Yaskawa INFORM job: A_ROOF_UPPER_0614_2_PAINT_28.JBI

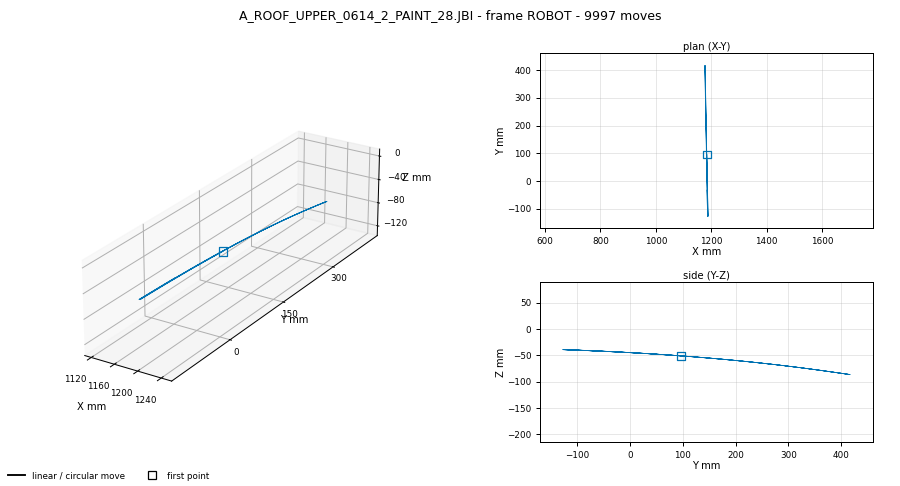
[picture p0: tool path of A_ROOF_UPPER_0614_2_PAINT_28.JBI in frame ROBOT, 9997 of 9997 moves have a stored position in this frame; points joined in program order, loops and branches not executed]
/JOB
//NAME A_ROOF_UPPER_0614_2_PAINT28
//POS
///NPOS 9997,0,0,0,0,0
///TOOL 1
///USER 0
///POSTYPE ROBOT
///RECTAN
///RCONF 1,0,0,0,0,0,0,0,0,0,0,0,0,0,0,0,0,0,0,0,0,0,0,0
C00000=1184.415,96.104,-50.756,-178.923,6.084,148.774
C00001=1184.420,95.856,-50.738,-178.925,6.082,148.774
C00002=1184.424,95.607,-50.720,-178.928,6.081,148.774
C00003=1184.429,95.357,-50.701,-178.931,6.080,148.775
C00004=1184.434,95.107,-50.683,-178.933,6.079,148.775
C00005=1184.439,94.858,-50.665,-178.936,6.078,148.776
C00006=1184.444,94.609,-50.647,-178.938,6.077,148.777
C00007=1184.449,94.360,-50.629,-178.941,6.076,148.777
C00008=1184.454,94.111,-50.611,-178.944,6.075,148.778
C00009=1184.458,93.861,-50.592,-178.947,6.073,148.778
C00010=1184.463,93.612,-50.574,-178.949,6.072,148.779
C00011=1184.468,93.362,-50.556,-178.952,6.071,148.779
C00012=1184.473,93.113,-50.538,-178.954,6.070,148.780
C00013=1184.478,92.864,-50.521,-178.957,6.068,148.780
C00014=1184.483,92.615,-50.503,-178.960,6.068,148.781
C00015=1184.488,92.366,-50.485,-178.962,6.066,148.781
C00016=1184.492,92.116,-50.466,-178.965,6.066,148.782
C00017=1184.497,91.867,-50.448,-178.968,6.064,148.782
C00018=1184.502,91.618,-50.430,-178.970,6.063,148.783
C00019=1184.507,91.368,-50.412,-178.973,6.062,148.783
C00020=1184.512,91.119,-50.394,-178.975,6.061,148.784
C00021=1184.517,90.869,-50.377,-178.978,6.060,148.784
C00022=1184.522,90.620,-50.359,-178.980,6.058,148.785
C00023=1184.527,90.371,-50.341,-178.983,6.058,148.785
C00024=1184.532,90.122,-50.323,-178.986,6.056,148.786
C00025=1184.537,89.873,-50.305,-178.988,6.056,148.787
C00026=1184.541,89.623,-50.287,-178.991,6.054,148.787
C00027=1184.546,89.374,-50.269,-178.994,6.053,148.788
C00028=1184.551,89.124,-50.252,-178.996,6.052,148.788
C00029=1184.556,88.875,-50.234,-178.999,6.051,148.789
C00030=1184.561,88.625,-50.216,-179.002,6.049,148.789
C00031=1184.566,88.376,-50.198,-179.004,6.049,148.790
C00032=1184.571,88.127,-50.180,-179.007,6.047,148.790
C00033=1184.576,87.877,-50.162,-179.010,6.046,148.791
C00034=1184.581,87.628,-50.144,-179.012,6.046,148.791
C00035=1184.586,87.379,-50.126,-179.015,6.044,148.792
C00036=1184.590,87.130,-50.109,-179.017,6.043,148.792
C00037=1184.595,86.881,-50.091,-179.020,6.042,148.793
C00038=1184.600,86.631,-50.074,-179.023,6.041,148.793
C00039=1184.605,86.382,-50.056,-179.025,6.039,148.794
C00040=1184.610,86.133,-50.038,-179.028,6.039,148.794
C00041=1184.615,85.883,-50.021,-179.031,6.037,148.795
C00042=1184.620,85.634,-50.003,-179.033,6.036,148.796
C00043=1184.625,85.385,-49.985,-179.035,6.036,148.796
C00044=1184.629,85.136,-49.967,-179.039,6.034,148.797
C00045=1184.634,84.886,-49.950,-179.041,6.033,148.797
C00046=1184.639,84.637,-49.932,-179.044,6.032,148.798
C00047=1184.644,84.388,-49.914,-179.046,6.031,148.798
C00048=1184.649,84.138,-49.897,-179.049,6.030,148.799
C00049=1184.654,83.889,-49.879,-179.051,6.029,148.799
C00050=1184.659,83.639,-49.862,-179.054,6.028,148.800
C00051=1184.664,83.390,-49.844,-179.057,6.027,148.800
C00052=1184.669,83.141,-49.826,-179.059,6.026,148.801
C00053=1184.674,82.891,-49.809,-179.062,6.024,148.801
C00054=1184.678,82.642,-49.791,-179.065,6.024,148.802
C00055=1184.683,82.392,-49.774,-179.067,6.023,148.802
C00056=1184.688,82.143,-49.756,-179.070,6.021,148.803
C00057=1184.693,81.894,-49.738,-179.072,6.021,148.803
C00058=1184.698,81.645,-49.722,-179.075,6.019,148.804
C00059=1184.702,81.395,-49.704,-179.078,6.018,148.805
C00060=1184.708,81.146,-49.686,-179.081,6.017,148.805
C00061=1184.713,80.877,-49.667,-179.083,6.016,148.806
C00062=1184.719,80.609,-49.649,-179.086,6.015,148.806
C00063=1184.723,80.341,-49.630,-179.089,6.014,148.807
C00064=1184.728,80.072,-49.611,-179.092,6.013,148.808
C00065=1184.734,79.823,-49.594,-179.094,6.012,148.808
C00066=1184.739,79.573,-49.576,-179.097,6.011,148.809
C00067=1184.743,79.324,-49.559,-179.099,6.010,148.809
C00068=1184.749,79.075,-49.542,-179.102,6.009,148.810
C00069=1184.754,78.826,-49.524,-179.105,6.007,148.810
C00070=1184.758,78.576,-49.508,-179.107,6.007,148.811
C00071=1184.763,78.327,-49.490,-179.110,6.005,148.811
C00072=1184.768,78.077,-49.472,-179.113,6.005,148.812
C00073=1184.773,77.828,-49.455,-179.115,6.004,148.812
C00074=1184.778,77.579,-49.438,-179.118,6.002,148.813
C00075=1184.783,77.329,-49.420,-179.120,6.001,148.813
C00076=1184.788,77.081,-49.403,-179.123,6.000,148.814
C00077=1184.793,76.831,-49.386,-179.126,5.999,148.814
C00078=1184.797,76.582,-49.369,-179.128,5.999,148.815
C00079=1184.802,76.332,-49.351,-179.131,5.997,148.816
C00080=1184.808,76.082,-49.334,-179.134,5.996,148.816
C00081=1184.812,75.833,-49.317,-179.136,5.995,148.817
C00082=1184.817,75.584,-49.300,-179.139,5.994,148.817
C00083=1184.822,75.335,-49.283,-179.141,5.993,148.818
C00084=1184.827,75.085,-49.266,-179.144,5.992,148.818
C00085=1184.831,74.836,-49.249,-179.146,5.991,148.819
C00086=1184.837,74.586,-49.231,-179.149,5.990,148.819
C00087=1184.842,74.337,-49.214,-179.152,5.989,148.820
C00088=1184.846,74.088,-49.197,-179.154,5.988,148.821
C00089=1184.852,73.839,-49.180,-179.157,5.988,148.821
C00090=1184.856,73.589,-49.163,-179.160,5.986,148.822
C00091=1184.862,73.339,-49.146,-179.162,5.985,148.822
C00092=1184.866,73.091,-49.128,-179.165,5.984,148.823
C00093=1184.871,72.841,-49.111,-179.168,5.983,148.823
C00094=1184.876,72.592,-49.095,-179.170,5.982,148.824
C00095=1184.881,72.342,-49.078,-179.173,5.981,148.824
C00096=1184.886,72.093,-49.061,-179.175,5.980,148.825
C00097=1184.891,71.843,-49.044,-179.178,5.979,148.826
C00098=1184.896,71.595,-49.027,-179.181,5.978,148.826
C00099=1184.901,71.345,-49.009,-179.183,5.977,148.827
C00100=1184.905,71.095,-48.993,-179.186,5.977,148.827
C00101=1184.911,70.846,-48.976,-179.189,5.975,148.828
C00102=1184.915,70.596,-48.959,-179.191,5.974,148.828
C00103=1184.921,70.347,-48.942,-179.193,5.974,148.829
C00104=1184.925,70.098,-48.925,-179.197,5.972,148.829
C00105=1184.930,69.848,-48.907,-179.199,5.971,148.830
C00106=1184.935,69.599,-48.891,-179.201,5.971,148.831
C00107=1184.940,69.350,-48.874,-179.204,5.969,148.831
C00108=1184.945,69.100,-48.857,-179.207,5.969,148.832
C00109=1184.950,68.851,-48.840,-179.209,5.968,148.832
C00110=1184.955,68.602,-48.823,-179.212,5.966,148.833
C00111=1184.960,68.352,-48.807,-179.215,5.966,148.833
C00112=1184.964,68.103,-48.790,-179.217,5.965,148.834
C00113=1184.970,67.853,-48.773,-179.220,5.964,148.835
C00114=1184.975,67.604,-48.757,-179.222,5.963,148.835
C00115=1184.980,67.354,-48.739,-179.225,5.962,148.836
C00116=1184.984,67.105,-48.723,-179.228,5.960,148.836
C00117=1184.990,66.856,-48.706,-179.230,5.960,148.837
C00118=1184.995,66.606,-48.689,-179.233,5.959,148.837
C00119=1184.999,66.357,-48.672,-179.236,5.958,148.838
C00120=1185.004,66.107,-48.656,-179.238,5.957,148.838
C00121=1185.010,65.858,-48.639,-179.240,5.956,148.839
C00122=1185.014,65.609,-48.622,-179.244,5.955,148.840
C00123=1185.018,65.359,-48.605,-179.246,5.954,148.840
C00124=1185.024,65.110,-48.589,-179.248,5.953,148.841
C00125=1185.029,64.861,-48.572,-179.252,5.952,148.841
C00126=1185.033,64.611,-48.555,-179.254,5.951,148.842
C00127=1185.039,64.362,-48.538,-179.256,5.951,148.842
C00128=1185.044,64.112,-48.522,-179.258,5.950,148.843
C00129=1185.049,63.863,-48.506,-179.262,5.948,148.843
C00130=1185.053,63.614,-48.489,-179.264,5.948,148.844
C00131=1185.059,63.364,-48.472,-179.266,5.947,148.845
C00132=1185.064,63.115,-48.456,-179.270,5.946,148.845
C00133=1185.068,62.866,-48.439,-179.272,5.945,148.846
C00134=1185.073,62.616,-48.423,-179.274,5.944,148.846
C00135=1185.079,62.367,-48.406,-179.277,5.943,148.847
C00136=1185.083,62.117,-48.390,-179.280,5.942,148.847
C00137=1185.088,61.868,-48.373,-179.282,5.941,148.848
C00138=1185.093,61.619,-48.357,-179.285,5.941,148.849
C00139=1185.098,61.369,-48.339,-179.288,5.939,148.849
C00140=1185.103,61.120,-48.324,-179.290,5.938,148.850
C00141=1185.108,60.870,-48.307,-179.293,5.938,148.850
C00142=1185.113,60.621,-48.291,-179.295,5.936,148.851
C00143=1185.117,60.372,-48.274,-179.298,5.936,148.851
C00144=1185.123,60.121,-48.258,-179.301,5.935,148.852
C00145=1185.128,59.873,-48.241,-179.303,5.934,148.853
C00146=1185.133,59.623,-48.225,-179.306,5.933,148.853
C00147=1185.138,59.374,-48.208,-179.308,5.932,148.854
C00148=1185.142,59.124,-48.192,-179.311,5.931,148.854
C00149=1185.148,58.875,-48.176,-179.313,5.931,148.855
C00150=1185.153,58.626,-48.159,-179.316,5.929,148.855
C00151=1185.158,58.376,-48.143,-179.319,5.929,148.856
C00152=1185.163,58.127,-48.127,-179.321,5.928,148.856
C00153=1185.167,57.877,-48.110,-179.324,5.927,148.857
C00154=1185.172,57.628,-48.094,-179.327,5.926,148.858
C00155=1185.177,57.378,-48.078,-179.329,5.925,148.858
C00156=1185.182,57.130,-48.061,-179.332,5.925,148.859
C00157=1185.188,56.879,-48.045,-179.334,5.923,148.859
C00158=1185.193,56.630,-48.029,-179.337,5.922,148.860
C00159=1185.197,56.380,-48.013,-179.340,5.922,148.861
C00160=1185.202,56.132,-47.996,-179.342,5.921,148.861
C00161=1185.207,55.882,-47.980,-179.345,5.920,148.862
C00162=1185.212,55.633,-47.964,-179.347,5.919,148.862
C00163=1185.217,55.383,-47.947,-179.350,5.918,148.863
C00164=1185.222,55.134,-47.932,-179.352,5.918,148.864
C00165=1185.227,54.865,-47.914,-179.355,5.916,148.864
C00166=1185.232,54.597,-47.897,-179.358,5.915,148.865
C00167=1185.238,54.328,-47.880,-179.361,5.914,148.865
C00168=1185.243,54.059,-47.861,-179.364,5.914,148.866
C00169=1185.249,53.810,-47.845,-179.366,5.913,148.866
C00170=1185.253,53.560,-47.829,-179.369,5.911,148.867
C00171=1185.259,53.311,-47.813,-179.372,5.911,148.868
C00172=1185.264,53.062,-47.797,-179.374,5.910,148.868
C00173=1185.269,52.812,-47.781,-179.376,5.909,148.869
C00174=1185.274,52.563,-47.765,-179.379,5.908,148.869
C00175=1185.278,52.313,-47.749,-179.382,5.907,148.870
C00176=1185.284,52.064,-47.733,-179.384,5.907,148.871
C00177=1185.288,51.814,-47.716,-179.386,5.906,148.871
C00178=1185.294,51.565,-47.701,-179.389,5.905,148.872
C00179=1185.298,51.316,-47.684,-179.392,5.904,148.872
C00180=1185.303,51.066,-47.668,-179.395,5.903,148.873
C00181=1185.308,50.818,-47.653,-179.397,5.903,148.874
C00182=1185.313,50.568,-47.637,-179.399,5.902,148.874
C00183=1185.318,50.318,-47.621,-179.403,5.900,148.875
C00184=1185.322,50.069,-47.605,-179.405,5.900,148.875
C00185=1185.328,49.819,-47.589,-179.407,5.899,148.876
C00186=1185.332,49.570,-47.572,-179.410,5.898,148.876
C00187=1185.338,49.320,-47.557,-179.413,5.898,148.877
C00188=1185.343,49.071,-47.541,-179.415,5.896,148.878
C00189=1185.348,48.822,-47.524,-179.418,5.896,148.878
C00190=1185.353,48.572,-47.509,-179.420,5.895,148.879
C00191=1185.358,48.322,-47.493,-179.423,5.894,148.879
C00192=1185.362,48.073,-47.478,-179.426,5.893,148.880
C00193=1185.368,47.824,-47.462,-179.428,5.892,148.880
C00194=1185.372,47.574,-47.446,-179.431,5.892,148.881
C00195=1185.378,47.325,-47.430,-179.433,5.891,148.882
C00196=1185.383,47.076,-47.414,-179.436,5.890,148.882
C00197=1185.388,46.826,-47.398,-179.439,5.889,148.883
C00198=1185.393,46.576,-47.382,-179.441,5.888,148.883
C00199=1185.398,46.326,-47.366,-179.444,5.888,148.884
C00200=1185.402,46.078,-47.351,-179.446,5.887,148.885
C00201=1185.407,45.828,-47.335,-179.448,5.886,148.885
C00202=1185.412,45.578,-47.319,-179.452,5.885,148.886
C00203=1185.418,45.329,-47.303,-179.454,5.884,148.886
C00204=1185.423,45.079,-47.288,-179.456,5.883,148.887
C00205=1185.427,44.830,-47.272,-179.459,5.883,148.888
C00206=1185.432,44.581,-47.256,-179.462,5.882,148.888
C00207=1185.438,44.331,-47.241,-179.464,5.881,148.889
C00208=1185.442,44.081,-47.225,-179.467,5.880,148.889
C00209=1185.448,43.832,-47.209,-179.469,5.879,148.890
C00210=1185.452,43.583,-47.194,-179.472,5.879,148.890
C00211=1185.457,43.334,-47.178,-179.474,5.878,148.891
C00212=1185.462,43.084,-47.162,-179.477,5.877,148.892
C00213=1185.468,42.835,-47.146,-179.480,5.876,148.892
C00214=1185.472,42.585,-47.131,-179.482,5.876,148.893
C00215=1185.477,42.335,-47.115,-179.485,5.875,148.893
C00216=1185.482,42.086,-47.100,-179.487,5.874,148.894
C00217=1185.488,41.837,-47.084,-179.490,5.874,148.895
C00218=1185.492,41.587,-47.069,-179.493,5.872,148.895
C00219=1185.497,41.337,-47.053,-179.495,5.871,148.896
C00220=1185.503,41.088,-47.038,-179.498,5.871,148.896
C00221=1185.508,40.839,-47.021,-179.500,5.870,148.897
C00222=1185.512,40.589,-47.006,-179.503,5.870,148.898
C00223=1185.517,40.340,-46.990,-179.505,5.869,148.898
C00224=1185.523,40.091,-46.975,-179.508,5.867,148.899
C00225=1185.527,39.842,-46.960,-179.511,5.867,148.899
C00226=1185.532,39.591,-46.944,-179.513,5.866,148.900
C00227=1185.537,39.342,-46.928,-179.516,5.865,148.900
C00228=1185.542,39.093,-46.913,-179.518,5.865,148.901
C00229=1185.547,38.844,-46.898,-179.520,5.864,148.902
C00230=1185.553,38.594,-46.882,-179.523,5.864,148.902
C00231=1185.557,38.344,-46.867,-179.526,5.862,148.903
C00232=1185.563,38.094,-46.852,-179.528,5.861,148.903
C00233=1185.568,37.845,-46.836,-179.531,5.861,148.904
C00234=1185.573,37.596,-46.821,-179.534,5.860,148.905
C00235=1185.577,37.346,-46.805,-179.536,5.860,148.905
C00236=1185.582,37.097,-46.790,-179.538,5.859,148.906
C00237=1185.587,36.847,-46.775,-179.542,5.858,148.907
C00238=1185.593,36.598,-46.759,-179.544,5.857,148.907
C00239=1185.597,36.349,-46.744,-179.546,5.856,148.908
C00240=1185.603,36.099,-46.729,-179.549,5.856,148.908
C00241=1185.607,35.850,-46.713,-179.551,5.855,148.909
C00242=1185.613,35.599,-46.698,-179.554,5.854,148.909
C00243=1185.618,35.350,-46.683,-179.557,5.854,148.910
C00244=1185.623,35.101,-46.668,-179.559,5.852,148.911
C00245=1185.628,34.852,-46.652,-179.562,5.852,148.911
C00246=1185.632,34.602,-46.637,-179.565,5.851,148.912
C00247=1185.637,34.352,-46.621,-179.567,5.850,148.912
C00248=1185.642,34.103,-46.607,-179.569,5.850,148.913
C00249=1185.648,33.853,-46.591,-179.572,5.849,148.914
C00250=1185.652,33.604,-46.576,-179.574,5.848,148.914
C00251=1185.658,33.355,-46.561,-179.577,5.848,148.915
C00252=1185.662,33.106,-46.546,-179.580,5.847,148.916
C00253=1185.668,32.855,-46.530,-179.582,5.846,148.916
C00254=1185.672,32.606,-46.515,-179.585,5.845,148.917
C00255=1185.678,32.356,-46.500,-179.588,5.845,148.917
C00256=1185.682,32.107,-46.485,-179.590,5.844,148.918
C00257=1185.688,31.857,-46.470,-179.592,5.843,148.918
C00258=1185.693,31.608,-46.455,-179.595,5.843,148.919
C00259=1185.698,31.359,-46.439,-179.597,5.842,148.920
C00260=1185.703,31.110,-46.424,-179.600,5.841,148.920
C00261=1185.708,30.860,-46.410,-179.603,5.840,148.921
C00262=1185.712,30.610,-46.394,-179.605,5.839,148.921
C00263=1185.718,30.361,-46.379,-179.608,5.839,148.922
C00264=1185.723,30.111,-46.364,-179.610,5.838,148.923
C00265=1185.728,29.861,-46.349,-179.613,5.838,148.923
C00266=1185.733,29.612,-46.334,-179.615,5.837,148.924
C00267=1185.738,29.363,-46.320,-179.618,5.836,148.925
C00268=1185.743,29.113,-46.304,-179.621,5.836,148.925
C00269=1185.748,28.844,-46.288,-179.623,5.834,148.926
C00270=1185.754,28.575,-46.272,-179.626,5.834,148.926
C00271=1185.759,28.307,-46.255,-179.629,5.833,148.927
C00272=1185.765,28.038,-46.239,-179.631,5.833,148.928
C00273=1185.770,27.788,-46.225,-179.634,5.831,148.928
C00274=1185.775,27.539,-46.209,-179.637,5.831,148.929
C00275=1185.780,27.290,-46.194,-179.639,5.830,148.930
C00276=1185.785,27.040,-46.180,-179.642,5.830,148.930
C00277=1185.790,26.791,-46.164,-179.645,5.829,148.931
C00278=1185.795,26.541,-46.150,-179.647,5.828,148.931
C00279=1185.800,26.292,-46.135,-179.649,5.828,148.932
C00280=1185.805,26.042,-46.120,-179.652,5.827,148.933
C00281=1185.810,25.793,-46.105,-179.654,5.826,148.933
C00282=1185.815,25.543,-46.091,-179.657,5.826,148.934
C00283=1185.820,25.294,-46.075,-179.659,5.825,148.934
C00284=1185.825,25.044,-46.061,-179.662,5.824,148.935
C00285=1185.830,24.795,-46.046,-179.665,5.823,148.936
C00286=1185.836,24.545,-46.031,-179.667,5.823,148.936
C00287=1185.840,24.296,-46.016,-179.670,5.822,148.937
C00288=1185.845,24.046,-46.002,-179.672,5.821,148.937
C00289=1185.851,23.797,-45.986,-179.675,5.821,148.938
C00290=1185.856,23.547,-45.972,-179.678,5.820,148.939
C00291=1185.860,23.298,-45.957,-179.680,5.820,148.939
C00292=1185.865,23.048,-45.943,-179.682,5.819,148.940
C00293=1185.871,22.798,-45.928,-179.685,5.819,148.941
C00294=1185.876,22.549,-45.913,-179.687,5.818,148.941
C00295=1185.880,22.299,-45.899,-179.690,5.817,148.942
C00296=1185.885,22.050,-45.884,-179.692,5.817,148.942
C00297=1185.891,21.800,-45.869,-179.695,5.816,148.943
C00298=1185.896,21.551,-45.855,-179.698,5.815,148.944
C00299=1185.900,21.301,-45.840,-179.701,5.814,148.944
C00300=1185.905,21.052,-45.825,-179.703,5.814,148.945
C00301=1185.911,20.802,-45.810,-179.705,5.813,148.945
C00302=1185.916,20.553,-45.796,-179.708,5.812,148.946
C00303=1185.921,20.303,-45.781,-179.711,5.812,148.947
C00304=1185.925,20.054,-45.766,-179.713,5.811,148.947
C00305=1185.930,19.804,-45.752,-179.715,5.810,148.948
C00306=1185.936,19.554,-45.737,-179.718,5.810,148.949
C00307=1185.941,19.304,-45.723,-179.720,5.809,148.949
C00308=1185.946,19.055,-45.708,-179.723,5.808,148.950
C00309=1185.951,18.806,-45.694,-179.726,5.808,148.950
C00310=1185.956,18.557,-45.680,-179.728,5.807,148.951
C00311=1185.961,18.308,-45.665,-179.730,5.807,148.951
C00312=1185.966,18.057,-45.650,-179.733,5.806,148.952
C00313=1185.971,17.808,-45.635,-179.736,5.806,148.953
C00314=1185.976,17.558,-45.621,-179.738,5.805,148.953
C00315=1185.981,17.309,-45.606,-179.740,5.804,148.954
C00316=1185.986,17.059,-45.592,-179.743,5.804,148.955
C00317=1185.991,16.810,-45.578,-179.745,5.803,148.955
C00318=1185.996,16.560,-45.563,-179.749,5.802,148.956
C00319=1186.002,16.311,-45.549,-179.751,5.801,148.956
C00320=1186.007,16.061,-45.534,-179.754,5.801,148.957
C00321=1186.012,15.812,-45.520,-179.756,5.800,148.958
C00322=1186.017,15.562,-45.505,-179.759,5.799,148.958
C00323=1186.022,15.312,-45.491,-179.761,5.799,148.959
C00324=1186.027,15.063,-45.477,-179.763,5.798,148.959
C00325=1186.031,14.813,-45.462,-179.766,5.797,148.960
C00326=1186.037,14.564,-45.448,-179.769,5.797,148.961
C00327=1186.042,14.315,-45.434,-179.771,5.796,148.962
C00328=1186.047,14.065,-45.419,-179.774,5.796,148.962
C00329=1186.052,13.815,-45.405,-179.776,5.795,148.963
C00330=1186.057,13.566,-45.391,-179.779,5.795,148.963
C00331=1186.062,13.316,-45.376,-179.781,5.794,148.964
C00332=1186.067,13.067,-45.363,-179.784,5.793,148.964
C00333=1186.073,12.817,-45.348,-179.786,5.793,148.965
C00334=1186.077,12.568,-45.333,-179.789,5.792,148.966
C00335=1186.082,12.318,-45.318,-179.791,5.791,148.966
C00336=1186.087,12.068,-45.304,-179.794,5.791,148.967
C00337=1186.093,11.819,-45.290,-179.796,5.791,148.968
C00338=1186.098,11.570,-45.276,-179.799,5.790,148.968
C00339=1186.103,11.320,-45.262,-179.801,5.789,148.969
C00340=1186.108,11.070,-45.247,-179.804,5.789,148.969
C00341=1186.113,10.821,-45.233,-179.807,5.788,148.970
C00342=1186.118,10.572,-45.219,-179.809,5.787,148.971
C00343=1186.123,10.322,-45.206,-179.811,5.787,148.971
C00344=1186.128,10.072,-45.191,-179.814,5.786,148.972
C00345=1186.132,9.823,-45.177,-179.816,5.786,148.972
C00346=1186.138,9.574,-45.163,-179.819,5.785,148.973
C00347=1186.143,9.324,-45.149,-179.821,5.785,148.974
C00348=1186.148,9.074,-45.135,-179.824,5.784,148.975
C00349=1186.153,8.825,-45.120,-179.826,5.783,148.975
C00350=1186.158,8.575,-45.106,-179.829,5.783,148.976
C00351=1186.163,8.326,-45.092,-179.832,5.782,148.976
C00352=1186.169,8.076,-45.078,-179.834,5.781,148.977
C00353=1186.174,7.826,-45.064,-179.836,5.781,148.977
C00354=1186.179,7.577,-45.050,-179.839,5.780,148.978
C00355=1186.184,7.327,-45.036,-179.842,5.780,148.979
C00356=1186.189,7.077,-45.022,-179.844,5.779,148.979
C00357=1186.193,6.828,-45.008,-179.847,5.779,148.980
C00358=1186.199,6.579,-44.994,-179.849,5.778,148.981
C00359=1186.204,6.329,-44.980,-179.852,5.778,148.981
C00360=1186.209,6.080,-44.966,-179.854,5.777,148.982
C00361=1186.214,5.829,-44.952,-179.857,5.776,148.983
C00362=1186.220,5.580,-44.938,-179.859,5.776,148.983
C00363=1186.225,5.330,-44.924,-179.861,5.775,148.984
C00364=1186.229,5.081,-44.910,-179.864,5.774,148.984
C00365=1186.234,4.832,-44.896,-179.867,5.774,148.985
C00366=1186.239,4.582,-44.882,-179.869,5.774,148.986
C00367=1186.245,4.332,-44.868,-179.872,5.773,148.986
C00368=1186.250,4.083,-44.855,-179.874,5.772,148.987
C00369=1186.255,3.833,-44.840,-179.877,5.772,148.988
C00370=1186.259,3.584,-44.827,-179.880,5.771,148.988
C00371=1186.265,3.335,-44.813,-179.882,5.770,148.989
C00372=1186.270,3.085,-44.799,-179.884,5.770,148.989
C00373=1186.275,2.815,-44.784,-179.887,5.769,148.990
C00374=1186.281,2.546,-44.769,-179.890,5.769,148.991
C00375=1186.287,2.278,-44.754,-179.892,5.768,148.991
C00376=1186.292,2.008,-44.739,-179.895,5.768,148.992
C00377=1186.297,1.758,-44.725,-179.897,5.767,148.993
C00378=1186.302,1.509,-44.712,-179.900,5.767,148.993
C00379=1186.307,1.260,-44.698,-179.902,5.766,148.994
C00380=1186.312,1.009,-44.684,-179.905,5.766,148.995
C00381=1186.318,0.760,-44.670,-179.907,5.765,148.995
C00382=1186.322,0.511,-44.656,-179.910,5.764,148.996
C00383=1186.327,0.260,-44.643,-179.913,5.764,148.997
C00384=1186.333,0.011,-44.629,-179.915,5.763,148.997
C00385=1186.338,-0.238,-44.615,-179.917,5.763,148.998
C00386=1186.342,-0.488,-44.602,-179.920,5.762,148.998
C00387=1186.348,-0.737,-44.588,-179.922,5.762,148.999
C00388=1186.353,-0.987,-44.574,-179.925,5.762,149.000
C00389=1186.358,-1.236,-44.561,-179.927,5.761,149.000
C00390=1186.363,-1.486,-44.547,-179.930,5.761,149.001
C00391=1186.368,-1.736,-44.532,-179.932,5.760,149.002
C00392=1186.373,-1.985,-44.520,-179.934,5.759,149.002
C00393=1186.378,-2.235,-44.506,-179.937,5.759,149.003
C00394=1186.384,-2.484,-44.492,-179.940,5.758,149.003
C00395=1186.388,-2.734,-44.479,-179.942,5.758,149.004
C00396=1186.394,-2.983,-44.465,-179.945,5.757,149.005
C00397=1186.399,-3.233,-44.451,-179.947,5.757,149.005
C00398=1186.403,-3.483,-44.437,-179.950,5.756,149.006
C00399=1186.409,-3.732,-44.424,-179.953,5.756,149.007
C00400=1186.414,-3.982,-44.410,-179.955,5.755,149.007
C00401=1186.419,-4.231,-44.397,-179.957,5.754,149.008
C00402=1186.424,-4.481,-44.383,-179.960,5.754,149.008
C00403=1186.430,-4.731,-44.370,-179.962,5.754,149.009
C00404=1186.434,-4.980,-44.356,-179.964,5.753,149.010
C00405=1186.440,-5.230,-44.343,-179.967,5.753,149.010
C00406=1186.444,-5.479,-44.329,-179.970,5.752,149.011
C00407=1186.449,-5.729,-44.316,-179.972,5.752,149.011
C00408=1186.455,-5.978,-44.302,-179.974,5.751,149.012
C00409=1186.460,-6.228,-44.289,-179.977,5.751,149.013
C00410=1186.465,-6.478,-44.276,-179.980,5.750,149.014
C00411=1186.470,-6.727,-44.262,-179.982,5.749,149.014
C00412=1186.476,-6.977,-44.249,-179.985,5.749,149.015
C00413=1186.480,-7.227,-44.235,-179.987,5.748,149.015
C00414=1186.486,-7.476,-44.222,-179.990,5.748,149.016
C00415=1186.491,-7.726,-44.208,-179.992,5.747,149.017
C00416=1186.496,-7.975,-44.195,-179.994,5.747,149.017
C00417=1186.501,-8.225,-44.182,-179.997,5.747,149.018
C00418=1186.506,-8.474,-44.168,-179.999,5.746,149.019
C00419=1186.511,-8.724,-44.155,179.998,5.746,149.019
C00420=1186.516,-8.973,-44.141,179.996,5.745,149.020
C00421=1186.521,-9.223,-44.128,179.993,5.745,149.020
C00422=1186.526,-9.473,-44.115,179.990,5.744,149.021
C00423=1186.531,-9.722,-44.101,179.988,5.743,149.022
C00424=1186.536,-9.972,-44.088,179.986,5.743,149.022
C00425=1186.542,-10.222,-44.075,179.983,5.742,149.023
C00426=1186.546,-10.471,-44.061,179.981,5.743,149.024
C00427=1186.552,-10.720,-44.048,179.979,5.742,149.024
C00428=1186.557,-10.970,-44.035,179.976,5.741,149.025
C00429=1186.562,-11.219,-44.021,179.973,5.741,149.026
C00430=1186.567,-11.469,-44.008,179.971,5.740,149.026
C00431=1186.573,-11.719,-43.995,179.969,5.740,149.027
C00432=1186.577,-11.969,-43.982,179.966,5.739,149.027
C00433=1186.583,-12.218,-43.968,179.963,5.739,149.028
C00434=1186.587,-12.468,-43.955,179.961,5.738,149.029
C00435=1186.592,-12.717,-43.943,179.958,5.737,149.029
C00436=1186.598,-12.967,-43.930,179.956,5.738,149.030
C00437=1186.602,-13.216,-43.916,179.954,5.737,149.031
C00438=1186.608,-13.466,-43.903,179.952,5.736,149.031
C00439=1186.613,-13.716,-43.890,179.949,5.736,149.032
C00440=1186.619,-13.966,-43.877,179.946,5.735,149.032
C00441=1186.624,-14.214,-43.863,179.944,5.735,149.033
C00442=1186.628,-14.464,-43.850,179.941,5.734,149.034
C00443=1186.634,-14.714,-43.837,179.939,5.734,149.034
C00444=1186.638,-14.964,-43.824,179.937,5.734,149.035
C00445=1186.644,-15.213,-43.811,179.934,5.734,149.036
C00446=1186.649,-15.463,-43.798,179.932,5.733,149.036
C00447=1186.654,-15.712,-43.785,179.929,5.732,149.037
C00448=1186.660,-15.962,-43.771,179.927,5.732,149.038
C00449=1186.664,-16.212,-43.758,179.924,5.731,149.038
C00450=1186.669,-16.461,-43.746,179.922,5.731,149.039
C00451=1186.675,-16.711,-43.733,179.919,5.730,149.039
C00452=1186.680,-16.961,-43.720,179.917,5.730,149.040
C00453=1186.685,-17.210,-43.707,179.914,5.730,149.041
C00454=1186.691,-17.460,-43.694,179.912,5.729,149.041
C00455=1186.695,-17.709,-43.680,179.909,5.729,149.042
C00456=1186.700,-17.959,-43.668,179.907,5.728,149.043
C00457=1186.706,-18.208,-43.654,179.904,5.728,149.043
C00458=1186.710,-18.458,-43.641,179.902,5.727,149.044
C00459=1186.715,-18.708,-43.629,179.899,5.726,149.045
C00460=1186.721,-18.957,-43.616,179.897,5.727,149.045
C00461=1186.726,-19.207,-43.603,179.895,5.726,149.046
C00462=1186.731,-19.457,-43.590,179.892,5.725,149.046
C00463=1186.736,-19.706,-43.577,179.890,5.725,149.047
C00464=1186.741,-19.956,-43.564,179.887,5.725,149.048
C00465=1186.746,-20.206,-43.551,179.885,5.724,149.048
C00466=1186.752,-20.455,-43.539,179.882,5.723,149.049
C00467=1186.757,-20.705,-43.525,179.880,5.724,149.050
C00468=1186.762,-20.955,-43.513,179.878,5.723,149.050
C00469=1186.767,-21.204,-43.500,179.875,5.722,149.051
C00470=1186.772,-21.454,-43.487,179.873,5.722,149.051
C00471=1186.777,-21.704,-43.474,179.870,5.721,149.052
C00472=1186.783,-21.953,-43.461,179.867,5.721,149.053
C00473=1186.788,-22.202,-43.449,179.866,5.721,149.053
C00474=1186.792,-22.452,-43.436,179.863,5.720,149.054
C00475=1186.798,-22.702,-43.422,179.860,5.720,149.055
C00476=1186.803,-22.951,-43.410,179.858,5.720,149.055
C00477=1186.808,-23.221,-43.396,179.855,5.719,149.056
C00478=1186.814,-23.491,-43.382,179.852,5.719,149.057
C00479=1186.820,-23.761,-43.369,179.850,5.718,149.058
C00480=1186.825,-24.030,-43.356,179.847,5.718,149.058
C00481=1186.831,-24.280,-43.342,179.845,5.717,149.059
C00482=1186.836,-24.529,-43.330,179.842,5.716,149.059
C00483=1186.840,-24.779,-43.317,179.840,5.717,149.060
C00484=1186.845,-25.029,-43.304,179.838,5.716,149.061
C00485=1186.851,-25.278,-43.292,179.835,5.715,149.061
C00486=1186.856,-25.527,-43.279,179.833,5.715,149.062
C00487=1186.861,-25.778,-43.266,179.830,5.715,149.063
C00488=1186.866,-26.028,-43.254,179.828,5.714,149.063
C00489=1186.872,-26.277,-43.241,179.826,5.714,149.064
C00490=1186.877,-26.526,-43.228,179.823,5.714,149.064
C00491=1186.881,-26.776,-43.215,179.821,5.713,149.065
C00492=1186.886,-27.025,-43.203,179.818,5.712,149.066
C00493=1186.892,-27.275,-43.191,179.816,5.712,149.066
C00494=1186.897,-27.525,-43.178,179.813,5.711,149.067
C00495=1186.903,-27.774,-43.165,179.811,5.712,149.068
C00496=1186.907,-28.024,-43.152,179.809,5.711,149.068
C00497=1186.913,-28.274,-43.140,179.806,5.710,149.069
C00498=1186.918,-28.524,-43.128,179.803,5.710,149.070
C00499=1186.923,-28.773,-43.115,179.801,5.710,149.070
C00500=1186.928,-29.022,-43.102,179.799,5.710,149.071
C00501=1186.933,-29.273,-43.090,179.797,5.709,149.071
C00502=1186.938,-29.522,-43.078,179.794,5.709,149.072
C00503=1186.943,-29.772,-43.065,179.791,5.708,149.073
C00504=1186.948,-30.021,-43.052,179.789,5.707,149.073
C00505=1186.954,-30.271,-43.041,179.787,5.708,149.074
C00506=1186.959,-30.520,-43.028,179.784,5.707,149.075
C00507=1186.963,-30.770,-43.015,179.782,5.707,149.075
C00508=1186.969,-31.020,-43.003,179.779,5.706,149.076
C00509=1186.974,-31.269,-42.990,179.777,5.706,149.077
C00510=1186.979,-31.519,-42.978,179.775,5.706,149.077
C00511=1186.984,-31.769,-42.966,179.772,5.705,149.078
C00512=1186.990,-32.018,-42.953,179.770,5.705,149.078
C00513=1186.995,-32.267,-42.941,179.767,5.704,149.079
C00514=1186.999,-32.518,-42.929,179.765,5.704,149.080
C00515=1187.005,-32.767,-42.916,179.762,5.704,149.081
C00516=1187.010,-33.017,-42.904,179.760,5.703,149.081
C00517=1187.015,-33.266,-42.891,179.758,5.703,149.082
C00518=1187.020,-33.516,-42.879,179.755,5.702,149.082
C00519=1187.026,-33.766,-42.867,179.753,5.701,149.083
C00520=1187.031,-34.015,-42.854,179.751,5.702,149.084
C00521=1187.036,-34.265,-42.842,179.748,5.701,149.084
C00522=1187.041,-34.514,-42.830,179.745,5.701,149.085
C00523=1187.046,-34.764,-42.817,179.743,5.700,149.085
C00524=1187.051,-35.014,-42.805,179.741,5.700,149.086
C00525=1187.056,-35.264,-42.792,179.738,5.700,149.087
C00526=1187.062,-35.514,-42.781,179.736,5.700,149.088
C00527=1187.067,-35.763,-42.768,179.734,5.699,149.088
C00528=1187.072,-36.013,-42.756,179.731,5.698,149.089
C00529=1187.078,-36.262,-42.743,179.728,5.698,149.089
C00530=1187.083,-36.512,-42.732,179.726,5.698,149.090
C00531=1187.088,-36.761,-42.719,179.724,5.697,149.091
C00532=1187.094,-37.011,-42.707,179.721,5.697,149.091
C00533=1187.099,-37.261,-42.694,179.719,5.696,149.092
C00534=1187.103,-37.510,-42.683,179.717,5.697,149.093
C00535=1187.109,-37.760,-42.671,179.714,5.696,149.093
C00536=1187.113,-38.010,-42.658,179.712,5.696,149.094
C00537=1187.118,-38.260,-42.646,179.709,5.695,149.095
C00538=1187.124,-38.509,-42.634,179.706,5.695,149.095
C00539=1187.129,-38.759,-42.622,179.705,5.695,149.096
C00540=1187.134,-39.009,-42.609,179.702,5.694,149.096
C00541=1187.140,-39.259,-42.597,179.700,5.694,149.097
C00542=1187.144,-39.508,-42.585,179.697,5.693,149.098
C00543=1187.150,-39.758,-42.574,179.695,5.693,149.098
C00544=1187.155,-40.007,-42.561,179.693,5.693,149.099
C00545=1187.160,-40.257,-42.549,179.690,5.692,149.100
C00546=1187.166,-40.507,-42.537,179.688,5.692,149.100
C00547=1187.171,-40.756,-42.525,179.686,5.692,149.101
C00548=1187.175,-41.006,-42.513,179.683,5.691,149.102
C00549=1187.181,-41.256,-42.501,179.680,5.691,149.102
C00550=1187.186,-41.505,-42.489,179.678,5.690,149.103
C00551=1187.191,-41.755,-42.477,179.676,5.691,149.103
C00552=1187.197,-42.004,-42.464,179.673,5.690,149.104
C00553=1187.201,-42.254,-42.453,179.671,5.690,149.105
C00554=1187.207,-42.504,-42.441,179.669,5.689,149.105
C00555=1187.212,-42.753,-42.429,179.667,5.689,149.106
C00556=1187.217,-43.003,-42.417,179.664,5.689,149.107
C00557=1187.222,-43.253,-42.405,179.661,5.688,149.107
C00558=1187.227,-43.503,-42.394,179.659,5.688,149.108
C00559=1187.233,-43.752,-42.381,179.657,5.688,149.109
C00560=1187.238,-44.002,-42.369,179.654,5.687,149.109
C00561=1187.243,-44.251,-42.358,179.652,5.687,149.110
C00562=1187.248,-44.501,-42.345,179.649,5.686,149.110
C00563=1187.253,-44.751,-42.333,179.647,5.687,149.111
C00564=1187.259,-45.001,-42.321,179.645,5.686,149.112
C00565=1187.263,-45.250,-42.310,179.643,5.685,149.112
C00566=1187.269,-45.499,-42.298,179.640,5.685,149.113
C00567=1187.274,-45.749,-42.286,179.638,5.685,149.114
C00568=1187.280,-45.999,-42.274,179.635,5.685,149.114
C00569=1187.285,-46.248,-42.263,179.633,5.684,149.115
C00570=1187.290,-46.498,-42.251,179.630,5.684,149.116
C00571=1187.295,-46.748,-42.238,179.628,5.684,149.116
C00572=1187.300,-46.997,-42.227,179.626,5.683,149.117
C00573=1187.305,-47.247,-42.215,179.623,5.683,149.118
C00574=1187.311,-47.497,-42.203,179.621,5.682,149.118
C00575=1187.315,-47.747,-42.192,179.619,5.683,149.119
C00576=1187.321,-47.996,-42.179,179.616,5.682,149.119
C00577=1187.326,-48.246,-42.167,179.614,5.681,149.120
C00578=1187.331,-48.496,-42.156,179.611,5.681,149.121
C00579=1187.337,-48.745,-42.145,179.609,5.681,149.122
C00580=1187.342,-48.995,-42.133,179.607,5.680,149.122
C00581=1187.347,-49.265,-42.120,179.604,5.680,149.123
C00582=1187.353,-49.536,-42.107,179.602,5.680,149.123
C00583=1187.359,-49.806,-42.095,179.599,5.679,149.124
C00584=1187.364,-50.076,-42.082,179.597,5.679,149.125
C00585=1187.369,-50.326,-42.071,179.594,5.679,149.126
C00586=1187.374,-50.576,-42.059,179.591,5.679,149.126
C00587=1187.380,-50.825,-42.047,179.589,5.678,149.127
C00588=1187.385,-51.074,-42.035,179.587,5.678,149.127
C00589=1187.390,-51.324,-42.023,179.585,5.678,149.128
C00590=1187.395,-51.574,-42.012,179.582,5.677,149.129
C00591=1187.400,-51.823,-42.000,179.580,5.677,149.129
C00592=1187.406,-52.073,-41.988,179.578,5.677,149.130
C00593=1187.410,-52.323,-41.977,179.575,5.676,149.131
C00594=1187.416,-52.572,-41.966,179.573,5.676,149.131
C00595=1187.421,-52.822,-41.954,179.571,5.676,149.132
C00596=1187.427,-53.072,-41.942,179.568,5.675,149.133
C00597=1187.431,-53.321,-41.931,179.565,5.675,149.133
C00598=1187.437,-53.571,-41.919,179.564,5.675,149.134
C00599=1187.441,-53.821,-41.908,179.561,5.675,149.134
C00600=1187.447,-54.070,-41.896,179.558,5.674,149.135
C00601=1187.452,-54.320,-41.885,179.556,5.673,149.136
C00602=1187.458,-54.570,-41.873,179.554,5.674,149.136
C00603=1187.463,-54.820,-41.861,179.551,5.673,149.137
C00604=1187.468,-55.069,-41.850,179.549,5.673,149.138
C00605=1187.473,-55.319,-41.838,179.547,5.673,149.138
C00606=1187.478,-55.568,-41.827,179.545,5.672,149.139
C00607=1187.484,-55.818,-41.815,179.542,5.672,149.140
C00608=1187.489,-56.068,-41.804,179.540,5.671,149.140
C00609=1187.494,-56.318,-41.793,179.538,5.672,149.141
C00610=1187.499,-56.568,-41.782,179.535,5.671,149.142
C00611=1187.504,-56.817,-41.771,179.532,5.671,149.142
C00612=1187.510,-57.067,-41.759,179.531,5.671,149.143
C00613=1187.514,-57.316,-41.747,179.528,5.670,149.143
C00614=1187.520,-57.566,-41.736,179.525,5.670,149.144
C00615=1187.524,-57.816,-41.724,179.523,5.670,149.145
C00616=1187.531,-58.065,-41.713,179.521,5.669,149.145
C00617=1187.535,-58.315,-41.701,179.518,5.669,149.146
C00618=1187.541,-58.565,-41.690,179.516,5.669,149.147
C00619=1187.546,-58.815,-41.679,179.514,5.668,149.147
C00620=1187.551,-59.064,-41.668,179.511,5.668,149.148
C00621=1187.556,-59.314,-41.656,179.509,5.668,149.149
C00622=1187.561,-59.564,-41.645,179.507,5.668,149.149
C00623=1187.566,-59.813,-41.633,179.505,5.667,149.150
C00624=1187.572,-60.063,-41.623,179.502,5.667,149.150
C00625=1187.578,-60.313,-41.611,179.500,5.667,149.151
C00626=1187.582,-60.563,-41.600,179.498,5.666,149.152
C00627=1187.587,-60.812,-41.588,179.495,5.666,149.152
C00628=1187.593,-61.061,-41.577,179.493,5.666,149.153
C00629=1187.598,-61.312,-41.566,179.491,5.665,149.154
C00630=1187.603,-61.561,-41.555,179.488,5.665,149.154
C00631=1187.608,-61.811,-41.543,179.486,5.665,149.155
C00632=1187.613,-62.060,-41.532,179.483,5.665,149.156
C00633=1187.619,-62.311,-41.521,179.481,5.664,149.156
C00634=1187.624,-62.560,-41.510,179.479,5.665,149.157
C00635=1187.629,-62.809,-41.499,179.476,5.664,149.158
C00636=1187.634,-63.059,-41.487,179.474,5.663,149.158
C00637=1187.639,-63.309,-41.476,179.472,5.664,149.159
C00638=1187.645,-63.558,-41.465,179.469,5.663,149.159
C00639=1187.650,-63.808,-41.454,179.467,5.663,149.160
C00640=1187.655,-64.059,-41.443,179.465,5.663,149.161
C00641=1187.660,-64.308,-41.432,179.462,5.662,149.161
C00642=1187.666,-64.557,-41.420,179.460,5.662,149.162
C00643=1187.671,-64.808,-41.410,179.458,5.662,149.162
C00644=1187.676,-65.057,-41.398,179.456,5.661,149.163
C00645=1187.682,-65.307,-41.387,179.453,5.661,149.164
C00646=1187.687,-65.557,-41.376,179.451,5.661,149.164
C00647=1187.691,-65.806,-41.365,179.449,5.661,149.165
C00648=1187.697,-66.055,-41.354,179.446,5.660,149.166
C00649=1187.702,-66.306,-41.343,179.444,5.661,149.167
C00650=1187.708,-66.555,-41.332,179.442,5.660,149.167
C00651=1187.712,-66.804,-41.321,179.439,5.659,149.168
C00652=1187.718,-67.055,-41.309,179.437,5.660,149.168
C00653=1187.723,-67.304,-41.298,179.435,5.659,149.169
C00654=1187.728,-67.554,-41.288,179.432,5.659,149.170
C00655=1187.733,-67.804,-41.277,179.430,5.659,149.170
C00656=1187.739,-68.053,-41.265,179.428,5.658,149.171
C00657=1187.744,-68.303,-41.255,179.425,5.658,149.171
C00658=1187.749,-68.553,-41.243,179.423,5.658,149.172
C00659=1187.754,-68.802,-41.233,179.420,5.658,149.173
C00660=1187.760,-69.052,-41.221,179.418,5.657,149.173
C00661=1187.765,-69.302,-41.211,179.416,5.657,149.174
C00662=1187.770,-69.552,-41.200,179.413,5.657,149.175
C00663=1187.775,-69.802,-41.189,179.411,5.656,149.175
C00664=1187.780,-70.051,-41.178,179.409,5.656,149.176
C00665=1187.786,-70.301,-41.167,179.407,5.656,149.177
C00666=1187.791,-70.550,-41.156,179.405,5.656,149.177
C00667=1187.796,-70.800,-41.145,179.402,5.655,149.178
C00668=1187.801,-71.050,-41.134,179.400,5.655,149.179
C00669=1187.807,-71.300,-41.124,179.398,5.655,149.179
C00670=1187.812,-71.550,-41.112,179.395,5.655,149.180
C00671=1187.818,-71.799,-41.102,179.393,5.654,149.180
C00672=1187.822,-72.049,-41.091,179.391,5.655,149.181
C00673=1187.828,-72.298,-41.080,179.388,5.654,149.182
C00674=1187.833,-72.548,-41.069,179.386,5.653,149.182
C00675=1187.838,-72.798,-41.059,179.384,5.654,149.183
C00676=1187.844,-73.047,-41.047,179.381,5.653,149.184
C00677=1187.849,-73.298,-41.036,179.379,5.653,149.184
C00678=1187.854,-73.547,-41.026,179.377,5.653,149.185
C00679=1187.859,-73.797,-41.015,179.375,5.652,149.185
C00680=1187.865,-74.046,-41.005,179.372,5.652,149.186
C00681=1187.869,-74.296,-40.993,179.370,5.652,149.187
C00682=1187.875,-74.545,-40.983,179.368,5.651,149.187
C00683=1187.880,-74.796,-40.973,179.365,5.652,149.188
C00684=1187.886,-75.045,-40.961,179.363,5.651,149.189
C00685=1187.891,-75.316,-40.950,179.360,5.651,149.189
C00686=1187.897,-75.587,-40.938,179.358,5.651,149.190
C00687=1187.903,-75.858,-40.926,179.356,5.650,149.191
C00688=1187.908,-76.129,-40.915,179.353,5.650,149.191
C00689=1187.913,-76.378,-40.904,179.351,5.650,149.192
C00690=1187.918,-76.628,-40.894,179.348,5.650,149.193
C00691=1187.923,-76.878,-40.883,179.346,5.649,149.193
C00692=1187.929,-77.127,-40.872,179.344,5.650,149.194
C00693=1187.934,-77.378,-40.861,179.342,5.649,149.195
C00694=1187.940,-77.627,-40.851,179.339,5.648,149.195
C00695=1187.945,-77.878,-40.840,179.337,5.649,149.196
C00696=1187.950,-78.126,-40.829,179.335,5.648,149.197
C00697=1187.956,-78.376,-40.819,179.332,5.647,149.197
C00698=1187.961,-78.626,-40.808,179.330,5.648,149.198
C00699=1187.966,-78.875,-40.798,179.328,5.647,149.198
C00700=1187.971,-79.125,-40.787,179.326,5.647,149.199
C00701=1187.977,-79.375,-40.777,179.323,5.647,149.200
C00702=1187.982,-79.625,-40.766,179.321,5.647,149.200
C00703=1187.987,-79.874,-40.755,179.319,5.647,149.201
C00704=1187.992,-80.124,-40.745,179.316,5.646,149.202
C00705=1187.998,-80.374,-40.734,179.314,5.647,149.202
C00706=1188.003,-80.624,-40.724,179.312,5.646,149.203
C00707=1188.008,-80.873,-40.713,179.309,5.645,149.203
C00708=1188.013,-81.123,-40.702,179.307,5.646,149.204
C00709=1188.019,-81.373,-40.692,179.305,5.645,149.205
C00710=1188.024,-81.623,-40.682,179.303,5.645,149.205
C00711=1188.029,-81.873,-40.671,179.300,5.645,149.206
C00712=1188.034,-82.122,-40.660,179.298,5.644,149.207
C00713=1188.039,-82.372,-40.650,179.296,5.645,149.207
C00714=1188.045,-82.621,-40.640,179.294,5.644,149.208
C00715=1188.050,-82.872,-40.629,179.292,5.644,149.208
C00716=1188.056,-83.121,-40.619,179.289,5.644,149.209
C00717=1188.061,-83.371,-40.608,179.287,5.643,149.210
C00718=1188.065,-83.620,-40.598,179.285,5.643,149.210
C00719=1188.071,-83.870,-40.588,179.282,5.643,149.211
C00720=1188.076,-84.120,-40.577,179.280,5.643,149.212
C00721=1188.081,-84.369,-40.567,179.278,5.642,149.212
C00722=1188.086,-84.620,-40.556,179.275,5.642,149.213
C00723=1188.092,-84.869,-40.546,179.273,5.642,149.214
C00724=1188.098,-85.119,-40.536,179.271,5.642,149.214
C00725=1188.103,-85.369,-40.525,179.269,5.642,149.215
C00726=1188.108,-85.618,-40.515,179.266,5.642,149.216
C00727=1188.113,-85.868,-40.504,179.264,5.641,149.216
C00728=1188.118,-86.117,-40.494,179.262,5.641,149.217
C00729=1188.123,-86.367,-40.484,179.259,5.641,149.217
C00730=1188.128,-86.617,-40.474,179.258,5.641,149.218
C00731=1188.134,-86.867,-40.463,179.255,5.640,149.219
C00732=1188.139,-87.117,-40.453,179.253,5.640,149.219
C00733=1188.145,-87.366,-40.443,179.251,5.640,149.220
C00734=1188.150,-87.616,-40.432,179.248,5.640,149.221
C00735=1188.154,-87.866,-40.422,179.247,5.640,149.221
C00736=1188.160,-88.115,-40.412,179.244,5.639,149.222
C00737=1188.166,-88.365,-40.402,179.242,5.640,149.222
C00738=1188.171,-88.615,-40.391,179.240,5.639,149.223
C00739=1188.176,-88.865,-40.381,179.237,5.638,149.224
C00740=1188.182,-89.114,-40.371,179.235,5.639,149.224
C00741=1188.186,-89.364,-40.361,179.233,5.638,149.225
C00742=1188.192,-89.614,-40.351,179.231,5.638,149.226
C00743=1188.197,-89.863,-40.341,179.228,5.638,149.226
C00744=1188.202,-90.114,-40.330,179.226,5.637,149.227
C00745=1188.208,-90.363,-40.320,179.224,5.638,149.227
C00746=1188.213,-90.612,-40.310,179.221,5.637,149.228
C00747=1188.218,-90.863,-40.300,179.219,5.637,149.229
C00748=1188.223,-91.112,-40.289,179.217,5.637,149.229
C00749=1188.229,-91.362,-40.279,179.215,5.637,149.230
C00750=1188.234,-91.612,-40.269,179.212,5.636,149.231
C00751=1188.239,-91.862,-40.260,179.210,5.636,149.231
C00752=1188.245,-92.111,-40.249,179.208,5.636,149.232
C00753=1188.250,-92.362,-40.239,179.205,5.636,149.232
C00754=1188.255,-92.611,-40.229,179.204,5.636,149.233
C00755=1188.260,-92.860,-40.219,179.201,5.635,149.234
C00756=1188.266,-93.110,-40.209,179.199,5.636,149.234
C00757=1188.271,-93.360,-40.198,179.197,5.635,149.235
C00758=1188.276,-93.610,-40.188,179.194,5.634,149.236
C00759=1188.281,-93.859,-40.178,179.192,5.635,149.236
C00760=1188.287,-94.110,-40.169,179.190,5.634,149.237
C00761=1188.292,-94.359,-40.158,179.188,5.634,149.237
C00762=1188.297,-94.609,-40.149,179.186,5.634,149.238
C00763=1188.303,-94.858,-40.139,179.184,5.634,149.239
C00764=1188.308,-95.108,-40.128,179.181,5.634,149.239
C00765=1188.313,-95.358,-40.118,179.179,5.634,149.240
C00766=1188.318,-95.608,-40.109,179.177,5.633,149.241
C00767=1188.324,-95.857,-40.099,179.174,5.633,149.241
C00768=1188.329,-96.108,-40.088,179.172,5.633,149.242
C00769=1188.334,-96.357,-40.079,179.170,5.632,149.243
C00770=1188.339,-96.606,-40.068,179.168,5.632,149.243
C00771=1188.345,-96.856,-40.059,179.165,5.632,149.244
C00772=1188.350,-97.106,-40.049,179.163,5.632,149.244
C00773=1188.355,-97.356,-40.039,179.161,5.632,149.245
C00774=1188.361,-97.605,-40.028,179.159,5.632,149.246
C00775=1188.366,-97.855,-40.020,179.157,5.631,149.246
C00776=1188.371,-98.106,-40.009,179.154,5.631,149.247
C00777=1188.376,-98.355,-39.999,179.152,5.631,149.248
C00778=1188.381,-98.604,-39.989,179.150,5.630,149.248
C00779=1188.387,-98.855,-39.980,179.148,5.631,149.249
C00780=1188.393,-99.104,-39.969,179.145,5.630,149.249
C00781=1188.397,-99.354,-39.959,179.144,5.630,149.250
C00782=1188.403,-99.604,-39.950,179.141,5.630,149.251
C00783=1188.408,-99.853,-39.940,179.139,5.630,149.251
C00784=1188.413,-100.103,-39.930,179.137,5.630,149.252
C00785=1188.419,-100.352,-39.920,179.135,5.630,149.253
C00786=1188.424,-100.603,-39.911,179.132,5.629,149.253
C00787=1188.429,-100.853,-39.900,179.130,5.629,149.254
C00788=1188.434,-101.102,-39.891,179.128,5.629,149.254
C00789=1188.440,-101.374,-39.880,179.125,5.628,149.255
C00790=1188.446,-101.646,-39.870,179.123,5.629,149.256
C00791=1188.452,-101.917,-39.859,179.121,5.628,149.256
C00792=1188.458,-102.189,-39.848,179.118,5.628,149.257
C00793=1188.463,-102.438,-39.839,179.116,5.628,149.258
C00794=1188.468,-102.688,-39.829,179.114,5.628,149.258
C00795=1188.473,-102.938,-39.819,179.112,5.628,149.259
C00796=1188.478,-103.188,-39.809,179.109,5.627,149.259
C00797=1188.484,-103.437,-39.800,179.107,5.628,149.260
C00798=1188.489,-103.687,-39.790,179.105,5.627,149.261
C00799=1188.494,-103.936,-39.780,179.103,5.626,149.261
C00800=1188.500,-104.186,-39.771,179.101,5.626,149.262
C00801=1188.506,-104.436,-39.761,179.098,5.626,149.263
C00802=1188.510,-104.687,-39.751,179.097,5.626,149.263
C00803=1188.516,-104.936,-39.741,179.094,5.626,149.264
C00804=1188.521,-105.186,-39.732,179.092,5.626,149.264
C00805=1188.527,-105.435,-39.722,179.090,5.625,149.265
C00806=1188.531,-105.685,-39.712,179.088,5.626,149.266
C00807=1188.537,-105.935,-39.703,179.085,5.625,149.266
C00808=1188.542,-106.184,-39.693,179.083,5.625,149.267
C00809=1188.547,-106.435,-39.684,179.081,5.625,149.268
C00810=1188.552,-106.684,-39.674,179.079,5.625,149.268
C00811=1188.557,-106.934,-39.665,179.076,5.624,149.269
C00812=1188.563,-107.184,-39.655,179.075,5.624,149.269
C00813=1188.568,-107.433,-39.646,179.072,5.624,149.270
C00814=1188.574,-107.683,-39.636,179.071,5.624,149.270
C00815=1188.579,-107.933,-39.627,179.068,5.624,149.271
C00816=1188.585,-108.182,-39.617,179.066,5.624,149.272
C00817=1188.590,-108.432,-39.608,179.064,5.623,149.272
C00818=1188.595,-108.682,-39.597,179.061,5.623,149.273
C00819=1188.601,-108.932,-39.589,179.059,5.623,149.274
C00820=1188.606,-109.182,-39.578,179.057,5.623,149.274
C00821=1188.611,-109.432,-39.569,179.055,5.623,149.275
C00822=1188.616,-109.682,-39.560,179.052,5.622,149.276
C00823=1188.621,-109.931,-39.550,179.050,5.623,149.276
C00824=1188.627,-110.181,-39.541,179.048,5.622,149.277
C00825=1188.632,-110.431,-39.531,179.046,5.622,149.277
C00826=1188.637,-110.680,-39.522,179.044,5.621,149.278
C00827=1188.643,-110.930,-39.513,179.042,5.622,149.279
C00828=1188.648,-111.180,-39.503,179.039,5.621,149.279
C00829=1188.653,-111.430,-39.494,179.037,5.621,149.280
C00830=1188.659,-111.679,-39.484,179.035,5.621,149.280
C00831=1188.664,-111.929,-39.475,179.033,5.621,149.281
C00832=1188.669,-112.179,-39.466,179.030,5.621,149.282
C00833=1188.675,-112.428,-39.456,179.029,5.621,149.282
C00834=1188.680,-112.678,-39.447,179.026,5.620,149.283
C00835=1188.686,-112.928,-39.437,179.025,5.620,149.283
C00836=1188.691,-113.178,-39.428,179.022,5.620,149.284
C00837=1188.696,-113.427,-39.419,179.020,5.620,149.285
C00838=1188.702,-113.677,-39.409,179.018,5.620,149.285
C00839=1188.707,-113.927,-39.400,179.016,5.620,149.286
C00840=1188.712,-114.177,-39.391,179.013,5.619,149.287
C00841=1188.718,-114.427,-39.381,179.012,5.619,149.287
C00842=1188.723,-114.676,-39.372,179.009,5.619,149.288
C00843=1188.728,-114.926,-39.363,179.007,5.619,149.288
C00844=1188.734,-115.176,-39.353,179.005,5.618,149.289
C00845=1188.739,-115.425,-39.344,179.003,5.619,149.290
C00846=1188.744,-115.675,-39.335,179.001,5.618,149.290
C00847=1188.750,-115.925,-39.325,178.998,5.618,149.291
C00848=1188.755,-116.175,-39.316,178.996,5.618,149.291
C00849=1188.760,-116.424,-39.307,178.994,5.618,149.292
C00850=1188.765,-116.674,-39.298,178.992,5.617,149.293
C00851=1188.771,-116.924,-39.288,178.990,5.618,149.293
C00852=1188.776,-117.174,-39.279,178.988,5.617,149.294
C00853=1188.781,-117.424,-39.270,178.986,5.617,149.294
C00854=1188.787,-117.674,-39.260,178.983,5.617,149.295
C00855=1188.792,-117.924,-39.252,178.981,5.617,149.296
C00856=1188.797,-118.173,-39.243,178.979,5.617,149.296
C00857=1188.802,-118.423,-39.233,178.977,5.617,149.297
C00858=1188.808,-118.673,-39.224,178.974,5.616,149.298
C00859=1188.813,-118.923,-39.215,178.973,5.616,149.298
C00860=1188.818,-119.173,-39.206,178.970,5.616,149.299
C00861=1188.823,-119.422,-39.197,178.968,5.616,149.299
C00862=1188.829,-119.672,-39.187,178.966,5.615,149.300
C00863=1188.834,-119.922,-39.178,178.964,5.615,149.300
C00864=1188.839,-120.172,-39.169,178.962,5.615,149.301
C00865=1188.844,-120.421,-39.160,178.960,5.615,149.302
C00866=1188.850,-120.671,-39.151,178.957,5.615,149.302
C00867=1188.855,-120.921,-39.142,178.956,5.615,149.303
C00868=1188.860,-121.171,-39.132,178.953,5.614,149.304
C00869=1188.865,-121.421,-39.123,178.951,5.614,149.304
C00870=1188.871,-121.670,-39.115,178.949,5.614,149.305
C00871=1188.876,-121.920,-39.106,178.947,5.614,149.305
C00872=1188.882,-122.170,-39.096,178.944,5.614,149.306
C00873=1188.887,-122.420,-39.087,178.943,5.614,149.306
C00874=1188.893,-122.669,-39.078,178.941,5.614,149.307
C00875=1188.898,-122.919,-39.069,178.939,5.613,149.308
C00876=1188.903,-123.169,-39.061,178.936,5.614,149.308
C00877=1188.909,-123.419,-39.050,178.934,5.613,149.309
C00878=1188.914,-123.669,-39.041,178.932,5.613,149.310
C00879=1188.919,-123.918,-39.033,178.930,5.613,149.310
C00880=1188.924,-124.168,-39.024,178.928,5.613,149.311
C00881=1188.930,-124.417,-39.015,178.926,5.612,149.311
C00882=1188.935,-124.667,-39.006,178.924,5.613,149.312
C00883=1188.940,-124.917,-38.997,178.921,5.612,149.312
C00884=1188.946,-125.167,-38.988,178.919,5.612,149.313
C00885=1188.951,-125.417,-38.979,178.917,5.611,149.314
C00886=1188.956,-125.667,-38.970,178.915,5.612,149.314
C00887=1188.962,-125.917,-38.961,178.913,5.611,149.315
C00888=1188.967,-126.167,-38.952,178.911,5.612,149.316
C00889=1188.973,-126.416,-38.944,178.909,5.611,149.316
C00890=1188.978,-126.666,-38.935,178.906,5.611,149.317
C00891=1188.983,-126.916,-38.926,178.904,5.610,149.317
C00892=1188.989,-127.166,-38.916,178.902,5.611,149.318
C00893=1188.567,-127.176,-38.956,178.898,5.614,149.320
C00894=1188.562,-126.926,-38.965,178.901,5.614,149.319
C00895=1188.556,-126.677,-38.974,178.903,5.614,149.319
C00896=1188.551,-126.427,-38.982,178.905,5.615,149.318
C00897=1188.546,-126.177,-38.991,178.907,5.615,149.317
C00898=1188.541,-125.927,-39.000,178.909,5.614,149.317
C00899=1188.534,-125.678,-39.009,178.911,5.615,149.316
C00900=1188.529,-125.428,-39.018,178.913,5.615,149.316
C00901=1188.524,-125.178,-39.027,178.915,5.615,149.315
C00902=1188.519,-124.928,-39.036,178.917,5.615,149.314
C00903=1188.514,-124.678,-39.045,178.920,5.616,149.314
C00904=1188.509,-124.429,-39.055,178.922,5.615,149.313
C00905=1188.504,-124.179,-39.063,178.924,5.616,149.313
C00906=1188.498,-123.929,-39.073,178.926,5.616,149.312
C00907=1188.492,-123.680,-39.081,178.928,5.617,149.311
C00908=1188.487,-123.430,-39.090,178.930,5.616,149.311
C00909=1188.482,-123.180,-39.099,178.933,5.617,149.310
C00910=1188.477,-122.930,-39.108,178.934,5.617,149.310
C00911=1188.471,-122.680,-39.117,178.937,5.617,149.309
C00912=1188.466,-122.431,-39.126,178.939,5.617,149.308
C00913=1188.460,-122.180,-39.135,178.941,5.618,149.308
C00914=1188.455,-121.931,-39.144,178.943,5.617,149.307
C00915=1188.450,-121.681,-39.153,178.945,5.618,149.307
C00916=1188.445,-121.431,-39.163,178.947,5.618,149.306
C00917=1188.440,-121.182,-39.172,178.950,5.618,149.305
C00918=1188.433,-120.932,-39.181,178.952,5.618,149.305
C00919=1188.428,-120.682,-39.190,178.954,5.619,149.304
C00920=1188.423,-120.432,-39.199,178.956,5.618,149.304
C00921=1188.418,-120.183,-39.208,178.958,5.618,149.303
C00922=1188.413,-119.933,-39.217,178.960,5.619,149.302
C00923=1188.407,-119.683,-39.227,178.962,5.619,149.302
C00924=1188.402,-119.433,-39.236,178.965,5.619,149.301
C00925=1188.397,-119.184,-39.245,178.966,5.619,149.301
C00926=1188.392,-118.934,-39.253,178.969,5.619,149.300
C00927=1188.386,-118.683,-39.263,178.970,5.619,149.299
C00928=1188.381,-118.434,-39.273,178.973,5.620,149.299
C00929=1188.376,-118.184,-39.281,178.975,5.620,149.298
C00930=1188.371,-117.935,-39.290,178.977,5.620,149.298
C00931=1188.365,-117.684,-39.300,178.979,5.620,149.297
C00932=1188.359,-117.435,-39.309,178.982,5.621,149.296
C00933=1188.355,-117.185,-39.318,178.983,5.621,149.296
C00934=1188.349,-116.935,-39.327,178.986,5.621,149.295
C00935=1188.344,-116.685,-39.337,178.988,5.621,149.295
C00936=1188.338,-116.435,-39.346,178.990,5.621,149.294
C00937=1188.334,-116.186,-39.355,178.992,5.621,149.293
C00938=1188.328,-115.936,-39.365,178.995,5.622,149.293
C00939=1188.322,-115.686,-39.374,178.996,5.622,149.292
C00940=1188.317,-115.436,-39.383,178.999,5.622,149.291
C00941=1188.312,-115.187,-39.393,179.001,5.622,149.291
C00942=1188.307,-114.937,-39.402,179.003,5.622,149.290
C00943=1188.301,-114.687,-39.411,179.005,5.622,149.290
C00944=1188.296,-114.438,-39.421,179.007,5.623,149.289
C00945=1188.291,-114.188,-39.430,179.009,5.622,149.288
C00946=1188.285,-113.938,-39.439,179.012,5.623,149.288
C00947=1188.280,-113.688,-39.449,179.014,5.623,149.287
C00948=1188.275,-113.438,-39.458,179.016,5.624,149.287
C00949=1188.270,-113.189,-39.467,179.018,5.623,149.286
C00950=1188.264,-112.939,-39.477,179.020,5.624,149.285
C00951=1188.259,-112.689,-39.486,179.022,5.623,149.285
C00952=1188.254,-112.439,-39.495,179.025,5.624,149.284
C00953=1188.248,-112.190,-39.505,179.027,5.624,149.284
C00954=1188.243,-111.940,-39.514,179.029,5.624,149.283
C00955=1188.237,-111.690,-39.523,179.031,5.624,149.282
C00956=1188.232,-111.441,-39.533,179.033,5.625,149.282
C00957=1188.227,-111.191,-39.542,179.035,5.625,149.281
C00958=1188.221,-110.941,-39.552,179.038,5.625,149.280
C00959=1188.216,-110.691,-39.561,179.040,5.626,149.280
C00960=1188.210,-110.441,-39.570,179.042,5.625,149.279
C00961=1188.205,-110.192,-39.580,179.044,5.626,149.279
C00962=1188.200,-109.942,-39.589,179.046,5.626,149.278
C00963=1188.195,-109.693,-39.599,179.049,5.626,149.277
C00964=1188.189,-109.443,-39.608,179.051,5.626,149.277
C00965=1188.184,-109.193,-39.618,179.053,5.627,149.276
C00966=1188.179,-108.943,-39.627,179.055,5.627,149.276
C00967=1188.174,-108.693,-39.636,179.058,5.627,149.275
C00968=1188.168,-108.443,-39.646,179.059,5.627,149.274
C00969=1188.163,-108.193,-39.655,179.062,5.627,149.274
C00970=1188.158,-107.944,-39.666,179.064,5.627,149.273
C00971=1188.153,-107.694,-39.674,179.066,5.628,149.273
C00972=1188.147,-107.444,-39.685,179.068,5.627,149.272
C00973=1188.142,-107.195,-39.694,179.070,5.628,149.271
C00974=1188.136,-106.945,-39.704,179.072,5.628,149.271
C00975=1188.131,-106.695,-39.713,179.075,5.628,149.270
C00976=1188.125,-106.446,-39.723,179.077,5.628,149.269
C00977=1188.121,-106.195,-39.732,179.079,5.628,149.269
C00978=1188.115,-105.946,-39.742,179.081,5.628,149.268
C00979=1188.110,-105.696,-39.751,179.084,5.629,149.268
C00980=1188.105,-105.446,-39.761,179.085,5.629,149.267
C00981=1188.099,-105.196,-39.770,179.088,5.629,149.266
C00982=1188.094,-104.947,-39.781,179.090,5.630,149.266
C00983=1188.089,-104.698,-39.790,179.092,5.630,149.265
C00984=1188.084,-104.447,-39.800,179.095,5.630,149.264
C00985=1188.079,-104.197,-39.810,179.097,5.630,149.264
C00986=1188.073,-103.947,-39.819,179.099,5.630,149.263
C00987=1188.068,-103.698,-39.829,179.101,5.630,149.263
C00988=1188.062,-103.448,-39.838,179.103,5.631,149.262
C00989=1188.057,-103.199,-39.848,179.106,5.630,149.261
C00990=1188.052,-102.949,-39.858,179.108,5.631,149.261
C00991=1188.047,-102.699,-39.867,179.110,5.631,149.260
C00992=1188.041,-102.449,-39.878,179.112,5.632,149.260
C00993=1188.037,-102.200,-39.887,179.114,5.631,149.259
C00994=1188.030,-101.928,-39.898,179.117,5.632,149.258
C00995=1188.024,-101.656,-39.908,179.119,5.632,149.258
C00996=1188.019,-101.385,-39.919,179.121,5.632,149.257
C00997=1188.013,-101.113,-39.930,179.124,5.632,149.256
C00998=1188.008,-100.864,-39.939,179.126,5.633,149.256
C00999=1188.002,-100.614,-39.949,179.128,5.633,149.255
C01000=1187.998,-100.363,-39.959,179.131,5.633,149.254
C01001=1187.992,-100.114,-39.969,179.133,5.633,149.254
C01002=1187.987,-99.864,-39.979,179.135,5.634,149.253
C01003=1187.981,-99.614,-39.988,179.137,5.633,149.252
C01004=1187.976,-99.365,-39.998,179.139,5.634,149.252
C01005=1187.972,-99.115,-40.008,179.141,5.634,149.251
C01006=1187.966,-98.865,-40.018,179.144,5.634,149.251
C01007=1187.960,-98.615,-40.028,179.146,5.635,149.250
C01008=1187.955,-98.366,-40.037,179.148,5.634,149.249
C01009=1187.950,-98.117,-40.048,179.150,5.635,149.249
C01010=1187.944,-97.866,-40.058,179.153,5.635,149.248
C01011=1187.939,-97.616,-40.067,179.155,5.635,149.247
C01012=1187.934,-97.367,-40.077,179.157,5.635,149.247
C01013=1187.928,-97.117,-40.088,179.159,5.635,149.246
C01014=1187.923,-96.868,-40.096,179.161,5.635,149.246
C01015=1187.918,-96.617,-40.107,179.164,5.636,149.245
C01016=1187.912,-96.368,-40.117,179.166,5.636,149.244
C01017=1187.908,-96.118,-40.127,179.168,5.636,149.244
C01018=1187.902,-95.869,-40.137,179.171,5.637,149.243
C01019=1187.897,-95.618,-40.147,179.172,5.637,149.243
C01020=1187.892,-95.369,-40.157,179.175,5.637,149.242
C01021=1187.886,-95.119,-40.167,179.177,5.637,149.241
C01022=1187.881,-94.870,-40.177,179.179,5.637,149.241
C01023=1187.876,-94.620,-40.187,179.181,5.637,149.240
C01024=1187.871,-94.370,-40.196,179.184,5.637,149.239
C01025=1187.865,-94.120,-40.207,179.186,5.638,149.239
C01026=1187.860,-93.870,-40.217,179.188,5.638,149.238
C01027=1187.855,-93.621,-40.227,179.190,5.639,149.238
C01028=1187.849,-93.371,-40.237,179.193,5.638,149.237
C01029=1187.844,-93.122,-40.247,179.195,5.639,149.236
C01030=1187.839,-92.871,-40.258,179.197,5.639,149.236
C01031=1187.834,-92.621,-40.267,179.200,5.639,149.235
C01032=1187.828,-92.372,-40.277,179.202,5.640,149.235
C01033=1187.823,-92.122,-40.288,179.204,5.639,149.234
C01034=1187.817,-91.872,-40.298,179.206,5.640,149.233
C01035=1187.813,-91.623,-40.307,179.208,5.640,149.233
C01036=1187.807,-91.373,-40.318,179.211,5.640,149.232
C01037=1187.802,-91.123,-40.328,179.213,5.640,149.231
C01038=1187.796,-90.874,-40.338,179.215,5.641,149.231
C01039=1187.792,-90.624,-40.348,179.218,5.641,149.230
C01040=1187.787,-90.374,-40.359,179.220,5.641,149.229
C01041=1187.781,-90.125,-40.369,179.222,5.641,149.229
C01042=1187.775,-89.875,-40.379,179.224,5.641,149.228
C01043=1187.770,-89.625,-40.390,179.226,5.642,149.228
C01044=1187.766,-89.376,-40.399,179.228,5.642,149.227
C01045=1187.760,-89.126,-40.409,179.231,5.642,149.226
C01046=1187.755,-88.876,-40.420,179.233,5.643,149.226
C01047=1187.749,-88.626,-40.430,179.235,5.642,149.225
C01048=1187.744,-88.377,-40.440,179.238,5.643,149.224
C01049=1187.739,-88.126,-40.451,179.240,5.643,149.224
C01050=1187.734,-87.877,-40.461,179.242,5.643,149.223
C01051=1187.728,-87.628,-40.471,179.245,5.644,149.222
C01052=1187.723,-87.377,-40.481,179.246,5.644,149.222
C01053=1187.718,-87.128,-40.492,179.249,5.644,149.221
C01054=1187.713,-86.878,-40.502,179.251,5.644,149.221
C01055=1187.707,-86.628,-40.512,179.253,5.644,149.220
C01056=1187.702,-86.379,-40.522,179.255,5.644,149.219
C01057=1187.697,-86.129,-40.532,179.258,5.645,149.219
C01058=1187.692,-85.879,-40.543,179.260,5.645,149.218
C01059=1187.687,-85.629,-40.553,179.262,5.645,149.217
C01060=1187.681,-85.379,-40.563,179.265,5.646,149.217
C01061=1187.675,-85.130,-40.574,179.267,5.645,149.216
C01062=1187.670,-84.879,-40.584,179.269,5.646,149.216
C01063=1187.665,-84.630,-40.594,179.272,5.646,149.215
C01064=1187.660,-84.380,-40.605,179.274,5.646,149.214
C01065=1187.655,-84.131,-40.615,179.276,5.646,149.214
C01066=1187.650,-83.882,-40.626,179.278,5.646,149.213
C01067=1187.645,-83.631,-40.636,179.281,5.647,149.212
C01068=1187.639,-83.382,-40.646,179.283,5.647,149.212
C01069=1187.634,-83.131,-40.657,179.285,5.647,149.211
C01070=1187.628,-82.882,-40.667,179.288,5.648,149.211
C01071=1187.623,-82.632,-40.677,179.289,5.648,149.210
C01072=1187.618,-82.383,-40.689,179.292,5.648,149.209
C01073=1187.613,-82.133,-40.699,179.294,5.648,149.209
C01074=1187.608,-81.883,-40.709,179.296,5.648,149.208
C01075=1187.602,-81.633,-40.720,179.299,5.649,149.207
C01076=1187.597,-81.383,-40.730,179.301,5.648,149.207
C01077=1187.592,-81.134,-40.741,179.303,5.649,149.206
C01078=1187.587,-80.884,-40.752,179.306,5.650,149.206
C01079=1187.581,-80.634,-40.762,179.308,5.649,149.205
C01080=1187.576,-80.385,-40.772,179.310,5.650,149.204
C01081=1187.571,-80.135,-40.783,179.312,5.650,149.204
C01082=1187.565,-79.886,-40.794,179.315,5.650,149.203
C01083=1187.560,-79.636,-40.804,179.317,5.651,149.202
C01084=1187.555,-79.386,-40.814,179.319,5.651,149.202
C01085=1187.550,-79.136,-40.825,179.322,5.651,149.201
C01086=1187.544,-78.887,-40.836,179.324,5.652,149.201
C01087=1187.539,-78.637,-40.846,179.326,5.651,149.200
C01088=1187.534,-78.387,-40.857,179.329,5.652,149.199
C01089=1187.529,-78.137,-40.867,179.330,5.652,149.199
C01090=1187.523,-77.888,-40.878,179.333,5.652,149.198
C01091=1187.518,-77.638,-40.889,179.336,5.653,149.197
C01092=1187.513,-77.388,-40.899,179.337,5.653,149.197
C01093=1187.508,-77.138,-40.910,179.340,5.653,149.196
C01094=1187.503,-76.889,-40.920,179.342,5.653,149.195
C01095=1187.498,-76.639,-40.931,179.344,5.653,149.195
C01096=1187.492,-76.390,-40.942,179.347,5.654,149.194
C01097=1187.487,-76.139,-40.953,179.349,5.654,149.193
C01098=1187.481,-75.869,-40.964,179.351,5.654,149.193
C01099=1187.475,-75.598,-40.976,179.354,5.654,149.192
C01100=1187.470,-75.327,-40.988,179.356,5.655,149.192
C01101=1187.464,-75.056,-40.999,179.358,5.655,149.191
C01102=1187.459,-74.806,-41.010,179.361,5.655,149.190
C01103=1187.453,-74.557,-41.020,179.364,5.656,149.189
C01104=1187.448,-74.307,-41.031,179.365,5.656,149.189
C01105=1187.442,-74.057,-41.042,179.368,5.656,149.188
C01106=1187.437,-73.807,-41.053,179.371,5.656,149.188
C01107=1187.432,-73.558,-41.064,179.372,5.656,149.187
C01108=1187.427,-73.308,-41.074,179.375,5.657,149.186
C01109=1187.422,-73.058,-41.085,179.377,5.656,149.186
C01110=1187.417,-72.809,-41.096,179.379,5.657,149.185
C01111=1187.412,-72.559,-41.107,179.382,5.658,149.184
C01112=1187.406,-72.309,-41.118,179.384,5.657,149.184
C01113=1187.401,-72.059,-41.129,179.387,5.658,149.183
C01114=1187.396,-71.810,-41.140,179.389,5.659,149.183
C01115=1187.391,-71.560,-41.150,179.391,5.658,149.182
C01116=1187.385,-71.311,-41.161,179.394,5.659,149.181
C01117=1187.380,-71.061,-41.172,179.396,5.659,149.181
C01118=1187.375,-70.811,-41.184,179.398,5.659,149.180
C01119=1187.369,-70.561,-41.194,179.401,5.659,149.179
C01120=1187.365,-70.312,-41.205,179.402,5.659,149.179
C01121=1187.359,-70.062,-41.215,179.405,5.660,149.178
C01122=1187.354,-69.812,-41.227,179.407,5.660,149.177
C01123=1187.349,-69.562,-41.238,179.409,5.660,149.177
C01124=1187.343,-69.313,-41.249,179.412,5.661,149.176
C01125=1187.338,-69.063,-41.259,179.414,5.661,149.175
C01126=1187.333,-68.814,-41.270,179.416,5.661,149.175
C01127=1187.328,-68.564,-41.281,179.419,5.662,149.174
C01128=1187.322,-68.314,-41.293,179.421,5.662,149.174
C01129=1187.317,-68.064,-41.303,179.423,5.662,149.173
C01130=1187.312,-67.814,-41.314,179.426,5.662,149.172
C01131=1187.307,-67.566,-41.325,179.428,5.663,149.172
C01132=1187.301,-67.315,-41.336,179.430,5.662,149.171
C01133=1187.296,-67.065,-41.347,179.433,5.663,149.170
C01134=1187.291,-66.816,-41.358,179.435,5.664,149.170
C01135=1187.285,-66.566,-41.370,179.437,5.663,149.169
C01136=1187.281,-66.316,-41.381,179.439,5.664,149.169
C01137=1187.275,-66.067,-41.391,179.442,5.665,149.168
C01138=1187.270,-65.817,-41.402,179.444,5.664,149.167
C01139=1187.265,-65.567,-41.414,179.446,5.665,149.167
C01140=1187.259,-65.318,-41.424,179.449,5.665,149.166
C01141=1187.255,-65.068,-41.436,179.451,5.665,149.165
C01142=1187.249,-64.817,-41.447,179.454,5.665,149.165
C01143=1187.244,-64.569,-41.458,179.456,5.666,149.164
C01144=1187.239,-64.319,-41.469,179.458,5.666,149.163
C01145=1187.234,-64.069,-41.480,179.461,5.666,149.163
C01146=1187.228,-63.819,-41.491,179.463,5.667,149.162
C01147=1187.223,-63.570,-41.502,179.465,5.667,149.162
C01148=1187.219,-63.320,-41.514,179.468,5.667,149.161
C01149=1187.212,-63.070,-41.525,179.470,5.668,149.160
C01150=1187.208,-62.821,-41.536,179.472,5.668,149.160
C01151=1187.202,-62.571,-41.548,179.475,5.668,149.159
C01152=1187.197,-62.321,-41.559,179.477,5.668,149.158
C01153=1187.192,-62.072,-41.569,179.479,5.668,149.158
C01154=1187.186,-61.822,-41.581,179.482,5.669,149.157
C01155=1187.182,-61.572,-41.592,179.484,5.669,149.156
C01156=1187.176,-61.323,-41.603,179.486,5.669,149.156
C01157=1187.171,-61.073,-41.615,179.488,5.670,149.155
C01158=1187.166,-60.823,-41.626,179.491,5.670,149.154
C01159=1187.161,-60.573,-41.637,179.493,5.670,149.154
C01160=1187.155,-60.324,-41.649,179.495,5.671,149.153
C01161=1187.150,-60.074,-41.659,179.498,5.671,149.153
C01162=1187.145,-59.824,-41.671,179.500,5.671,149.152
C01163=1187.140,-59.574,-41.682,179.502,5.671,149.151
C01164=1187.134,-59.325,-41.694,179.505,5.672,149.151
C01165=1187.129,-59.075,-41.705,179.508,5.672,149.150
C01166=1187.125,-58.826,-41.716,179.509,5.672,149.149
C01167=1187.119,-58.575,-41.728,179.512,5.673,149.149
C01168=1187.114,-58.326,-41.739,179.515,5.673,149.148
C01169=1187.108,-58.076,-41.750,179.517,5.673,149.147
C01170=1187.104,-57.827,-41.762,179.519,5.674,149.147
C01171=1187.098,-57.577,-41.774,179.522,5.674,149.146
C01172=1187.093,-57.328,-41.785,179.524,5.674,149.145
C01173=1187.088,-57.078,-41.796,179.526,5.675,149.145
C01174=1187.082,-56.828,-41.807,179.528,5.675,149.144
C01175=1187.078,-56.578,-41.818,179.531,5.675,149.144
C01176=1187.072,-56.328,-41.830,179.533,5.675,149.143
C01177=1187.067,-56.079,-41.841,179.535,5.676,149.142
C01178=1187.062,-55.829,-41.853,179.538,5.676,149.142
C01179=1187.057,-55.580,-41.864,179.540,5.676,149.141
C01180=1187.052,-55.330,-41.876,179.542,5.677,149.141
C01181=1187.047,-55.080,-41.887,179.545,5.677,149.140
C01182=1187.041,-54.831,-41.899,179.547,5.677,149.139
C01183=1187.036,-54.581,-41.910,179.550,5.677,149.138
C01184=1187.031,-54.331,-41.922,179.552,5.678,149.138
C01185=1187.026,-54.082,-41.933,179.554,5.678,149.137
C01186=1187.021,-53.832,-41.945,179.557,5.678,149.137
C01187=1187.016,-53.582,-41.957,179.559,5.679,149.136
C01188=1187.010,-53.333,-41.968,179.562,5.679,149.135
C01189=1187.005,-53.083,-41.979,179.564,5.679,149.135
C01190=1187.000,-52.833,-41.991,179.566,5.679,149.134
C01191=1186.994,-52.583,-42.003,179.568,5.680,149.133
C01192=1186.990,-52.334,-42.014,179.571,5.680,149.133
C01193=1186.984,-52.084,-42.026,179.573,5.680,149.132
C01194=1186.979,-51.835,-42.037,179.576,5.681,149.131
C01195=1186.973,-51.585,-42.049,179.578,5.682,149.131
C01196=1186.969,-51.335,-42.060,179.580,5.681,149.130
C01197=1186.963,-51.085,-42.072,179.583,5.682,149.129
C01198=1186.958,-50.835,-42.084,179.585,5.682,149.129
C01199=1186.953,-50.586,-42.096,179.588,5.683,149.128
C01200=1186.948,-50.336,-42.107,179.590,5.682,149.128
C01201=1186.943,-50.086,-42.119,179.592,5.683,149.127
C01202=1186.937,-49.817,-42.131,179.595,5.683,149.126
C01203=1186.932,-49.546,-42.144,179.597,5.684,149.126
C01204=1186.926,-49.277,-42.157,179.600,5.685,149.125
C01205=1186.920,-49.005,-42.170,179.602,5.684,149.124
C01206=1186.915,-48.756,-42.182,179.605,5.685,149.124
C01207=1186.910,-48.506,-42.194,179.607,5.685,149.123
C01208=1186.905,-48.257,-42.205,179.610,5.686,149.122
C01209=1186.900,-48.007,-42.217,179.612,5.686,149.122
C01210=1186.894,-47.757,-42.229,179.614,5.686,149.121
C01211=1186.889,-47.508,-42.240,179.617,5.686,149.120
C01212=1186.883,-47.258,-42.251,179.619,5.687,149.120
C01213=1186.878,-47.009,-42.264,179.621,5.687,149.119
C01214=1186.873,-46.759,-42.276,179.624,5.687,149.118
C01215=1186.868,-46.509,-42.287,179.626,5.688,149.118
C01216=1186.863,-46.259,-42.299,179.629,5.689,149.117
C01217=1186.857,-46.009,-42.311,179.631,5.688,149.117
C01218=1186.853,-45.760,-42.323,179.633,5.689,149.116
C01219=1186.848,-45.510,-42.335,179.636,5.689,149.115
C01220=1186.842,-45.260,-42.347,179.638,5.689,149.115
C01221=1186.837,-45.011,-42.358,179.640,5.690,149.114
C01222=1186.832,-44.761,-42.371,179.643,5.690,149.113
C01223=1186.827,-44.511,-42.383,179.645,5.691,149.113
C01224=1186.821,-44.262,-42.394,179.647,5.690,149.112
C01225=1186.817,-44.012,-42.406,179.650,5.691,149.111
C01226=1186.812,-43.763,-42.418,179.653,5.691,149.111
C01227=1186.806,-43.513,-42.430,179.655,5.692,149.110
C01228=1186.800,-43.263,-42.442,179.657,5.692,149.110
C01229=1186.796,-43.014,-42.454,179.659,5.692,149.109
C01230=1186.790,-42.764,-42.466,179.662,5.693,149.108
C01231=1186.785,-42.515,-42.478,179.664,5.694,149.108
C01232=1186.780,-42.265,-42.490,179.666,5.693,149.107
C01233=1186.774,-42.015,-42.502,179.669,5.694,149.106
C01234=1186.770,-41.766,-42.513,179.671,5.694,149.106
C01235=1186.765,-41.516,-42.526,179.674,5.695,149.105
C01236=1186.759,-41.266,-42.538,179.677,5.695,149.104
C01237=1186.754,-41.016,-42.550,179.679,5.695,149.104
C01238=1186.749,-40.767,-42.562,179.681,5.696,149.103
C01239=1186.744,-40.518,-42.574,179.684,5.696,149.103
C01240=1186.738,-40.268,-42.585,179.686,5.697,149.102
C01241=1186.733,-40.018,-42.598,179.688,5.696,149.101
C01242=1186.728,-39.768,-42.610,179.690,5.697,149.101
C01243=1186.723,-39.519,-42.623,179.693,5.698,149.100
C01244=1186.718,-39.268,-42.635,179.696,5.698,149.099
C01245=1186.713,-39.019,-42.646,179.698,5.698,149.099
C01246=1186.708,-38.769,-42.659,179.700,5.698,149.098
C01247=1186.703,-38.519,-42.671,179.703,5.699,149.097
C01248=1186.698,-38.270,-42.683,179.705,5.699,149.097
C01249=1186.692,-38.020,-42.695,179.708,5.700,149.096
C01250=1186.687,-37.771,-42.708,179.710,5.700,149.095
C01251=1186.682,-37.521,-42.720,179.712,5.700,149.095
C01252=1186.677,-37.272,-42.732,179.715,5.701,149.094
C01253=1186.672,-37.022,-42.743,179.717,5.702,149.094
C01254=1186.667,-36.773,-42.756,179.719,5.701,149.093
C01255=1186.661,-36.523,-42.768,179.722,5.702,149.092
C01256=1186.656,-36.273,-42.781,179.725,5.702,149.092
C01257=1186.651,-36.024,-42.792,179.727,5.703,149.091
C01258=1186.646,-35.774,-42.805,179.729,5.703,149.090
C01259=1186.640,-35.524,-42.817,179.731,5.703,149.090
C01260=1186.635,-35.275,-42.829,179.734,5.703,149.089
C01261=1186.630,-35.025,-42.841,179.736,5.704,149.088
C01262=1186.625,-34.775,-42.854,179.739,5.705,149.088
C01263=1186.620,-34.525,-42.866,179.741,5.704,149.087
C01264=1186.615,-34.276,-42.879,179.744,5.705,149.086
C01265=1186.609,-34.026,-42.891,179.746,5.706,149.086
C01266=1186.604,-33.776,-42.903,179.749,5.706,149.085
C01267=1186.599,-33.527,-42.916,179.751,5.707,149.085
C01268=1186.593,-33.277,-42.928,179.753,5.707,149.084
C01269=1186.588,-33.028,-42.940,179.755,5.707,149.083
C01270=1186.583,-32.778,-42.952,179.758,5.707,149.083
C01271=1186.578,-32.528,-42.965,179.761,5.708,149.082
C01272=1186.573,-32.279,-42.978,179.763,5.709,149.081
C01273=1186.568,-32.029,-42.990,179.765,5.708,149.081
C01274=1186.563,-31.779,-43.002,179.768,5.709,149.080
C01275=1186.558,-31.530,-43.015,179.770,5.709,149.079
C01276=1186.552,-31.280,-43.027,179.772,5.710,149.079
C01277=1186.547,-31.031,-43.039,179.775,5.711,149.078
C01278=1186.542,-30.781,-43.052,179.777,5.710,149.078
C01279=1186.537,-30.531,-43.064,179.780,5.711,149.077
C01280=1186.532,-30.282,-43.077,179.782,5.712,149.076
C01281=1186.527,-30.032,-43.089,179.785,5.712,149.076
C01282=1186.521,-29.782,-43.101,179.787,5.712,149.075
C01283=1186.516,-29.533,-43.114,179.790,5.713,149.074
C01284=1186.512,-29.283,-43.127,179.792,5.713,149.074
C01285=1186.506,-29.033,-43.139,179.794,5.713,149.073
C01286=1186.501,-28.784,-43.151,179.797,5.714,149.072
C01287=1186.496,-28.534,-43.164,179.800,5.714,149.072
C01288=1186.491,-28.285,-43.177,179.802,5.715,149.071
C01289=1186.486,-28.034,-43.189,179.804,5.715,149.071
C01290=1186.481,-27.785,-43.201,179.807,5.715,149.070
C01291=1186.476,-27.536,-43.214,179.809,5.716,149.069
C01292=1186.470,-27.286,-43.227,179.811,5.716,149.069
C01293=1186.465,-27.037,-43.240,179.814,5.717,149.068
C01294=1186.460,-26.786,-43.252,179.817,5.717,149.067
C01295=1186.455,-26.537,-43.265,179.818,5.717,149.067
C01296=1186.450,-26.288,-43.277,179.821,5.718,149.066
C01297=1186.445,-26.038,-43.290,179.824,5.718,149.065
C01298=1186.440,-25.789,-43.303,179.826,5.719,149.065
C01299=1186.435,-25.538,-43.315,179.828,5.720,149.064
C01300=1186.429,-25.289,-43.328,179.831,5.719,149.064
C01301=1186.424,-25.039,-43.341,179.833,5.720,149.063
C01302=1186.419,-24.790,-43.353,179.836,5.720,149.062
C01303=1186.414,-24.540,-43.366,179.838,5.721,149.062
C01304=1186.409,-24.291,-43.379,179.841,5.721,149.061
C01305=1186.404,-24.041,-43.391,179.843,5.722,149.060
C01306=1186.398,-23.771,-43.406,179.846,5.722,149.060
C01307=1186.393,-23.501,-43.419,179.849,5.723,149.059
C01308=1186.386,-23.232,-43.432,179.851,5.723,149.058
C01309=1186.381,-22.962,-43.446,179.854,5.724,149.057
C01310=1186.376,-22.713,-43.459,179.856,5.724,149.057
C01311=1186.370,-22.463,-43.472,179.858,5.724,149.056
C01312=1186.366,-22.213,-43.485,179.861,5.725,149.056
C01313=1186.361,-21.964,-43.498,179.864,5.725,149.055
C01314=1186.356,-21.714,-43.510,179.866,5.726,149.054
C01315=1186.351,-21.464,-43.523,179.868,5.726,149.054
C01316=1186.345,-21.215,-43.536,179.871,5.727,149.053
C01317=1186.340,-20.965,-43.549,179.873,5.727,149.052
C01318=1186.335,-20.716,-43.561,179.875,5.727,149.052
C01319=1186.331,-20.466,-43.574,179.878,5.728,149.051
C01320=1186.325,-20.216,-43.588,179.881,5.728,149.051
C01321=1186.320,-19.967,-43.600,179.883,5.729,149.050
C01322=1186.315,-19.717,-43.613,179.885,5.730,149.049
C01323=1186.309,-19.467,-43.626,179.888,5.730,149.049
C01324=1186.304,-19.218,-43.639,179.890,5.730,149.048
C01325=1186.299,-18.968,-43.652,179.893,5.730,149.047
C01326=1186.294,-18.719,-43.665,179.895,5.731,149.047
C01327=1186.289,-18.469,-43.678,179.898,5.731,149.046
C01328=1186.284,-18.219,-43.691,179.900,5.732,149.045
C01329=1186.279,-17.970,-43.703,179.903,5.732,149.045
C01330=1186.273,-17.720,-43.717,179.905,5.733,149.044
C01331=1186.268,-17.470,-43.730,179.907,5.733,149.044
C01332=1186.263,-17.221,-43.742,179.910,5.733,149.043
C01333=1186.258,-16.972,-43.756,179.912,5.734,149.042
C01334=1186.253,-16.722,-43.769,179.915,5.735,149.042
C01335=1186.248,-16.473,-43.782,179.917,5.735,149.041
C01336=1186.242,-16.223,-43.795,179.920,5.736,149.040
C01337=1186.238,-15.973,-43.808,179.922,5.736,149.040
C01338=1186.233,-15.724,-43.820,179.925,5.737,149.039
C01339=1186.227,-15.473,-43.834,179.927,5.737,149.038
C01340=1186.223,-15.225,-43.847,179.930,5.737,149.038
C01341=1186.217,-14.975,-43.860,179.932,5.738,149.037
C01342=1186.212,-14.725,-43.873,179.934,5.738,149.037
C01343=1186.207,-14.476,-43.886,179.937,5.739,149.036
C01344=1186.201,-14.226,-43.899,179.940,5.739,149.035
C01345=1186.197,-13.976,-43.912,179.942,5.740,149.035
C01346=1186.191,-13.727,-43.926,179.945,5.741,149.034
C01347=1186.187,-13.477,-43.939,179.947,5.740,149.033
C01348=1186.181,-13.228,-43.952,179.949,5.741,149.033
C01349=1186.176,-12.977,-43.965,179.951,5.742,149.032
C01350=1186.171,-12.729,-43.979,179.954,5.742,149.032
C01351=1186.166,-12.479,-43.992,179.957,5.742,149.031
C01352=1186.161,-12.229,-44.005,179.959,5.743,149.030
C01353=1186.155,-11.979,-44.018,179.962,5.744,149.030
C01354=1186.151,-11.730,-44.032,179.964,5.744,149.029
C01355=1186.145,-11.480,-44.045,179.967,5.745,149.028
C01356=1186.141,-11.230,-44.058,179.969,5.746,149.028
C01357=1186.135,-10.981,-44.070,179.971,5.745,149.027
C01358=1186.130,-10.732,-44.084,179.974,5.746,149.026
C01359=1186.125,-10.482,-44.097,179.976,5.746,149.026
C01360=1186.119,-10.232,-44.110,179.979,5.747,149.025
C01361=1186.115,-9.983,-44.124,179.981,5.747,149.025
C01362=1186.109,-9.733,-44.137,179.984,5.748,149.024
C01363=1186.105,-9.483,-44.150,179.987,5.748,149.023
C01364=1186.099,-9.234,-44.164,179.989,5.749,149.023
C01365=1186.095,-8.984,-44.177,179.991,5.750,149.022
C01366=1186.089,-8.735,-44.190,179.994,5.750,149.021
C01367=1186.085,-8.485,-44.204,179.996,5.750,149.021
C01368=1186.079,-8.235,-44.217,179.998,5.751,149.020
C01369=1186.075,-7.986,-44.231,-179.999,5.751,149.020
C01370=1186.069,-7.736,-44.244,-179.996,5.752,149.019
C01371=1186.064,-7.486,-44.258,-179.994,5.752,149.018
C01372=1186.059,-7.237,-44.271,-179.992,5.753,149.018
C01373=1186.053,-6.987,-44.284,-179.989,5.753,149.017
C01374=1186.049,-6.738,-44.298,-179.986,5.754,149.016
C01375=1186.043,-6.488,-44.311,-179.984,5.755,149.016
C01376=1186.039,-6.239,-44.325,-179.981,5.755,149.015
C01377=1186.033,-5.989,-44.338,-179.979,5.756,149.014
C01378=1186.027,-5.739,-44.351,-179.976,5.756,149.014
C01379=1186.023,-5.490,-44.365,-179.974,5.756,149.013
C01380=1186.017,-5.240,-44.378,-179.972,5.757,149.013
C01381=1186.013,-4.991,-44.392,-179.969,5.757,149.012
C01382=1186.008,-4.741,-44.406,-179.967,5.758,149.011
C01383=1186.002,-4.492,-44.419,-179.964,5.758,149.011
C01384=1185.998,-4.242,-44.432,-179.962,5.759,149.010
C01385=1185.992,-3.993,-44.446,-179.959,5.759,149.009
C01386=1185.988,-3.743,-44.459,-179.956,5.760,149.009
C01387=1185.982,-3.494,-44.473,-179.954,5.761,149.008
C01388=1185.977,-3.244,-44.488,-179.952,5.761,149.008
C01389=1185.972,-2.995,-44.500,-179.949,5.762,149.007
C01390=1185.967,-2.745,-44.514,-179.947,5.762,149.006
C01391=1185.962,-2.495,-44.528,-179.944,5.763,149.006
C01392=1185.957,-2.246,-44.541,-179.941,5.763,149.005
C01393=1185.952,-1.996,-44.555,-179.939,5.764,149.004
C01394=1185.946,-1.746,-44.569,-179.937,5.765,149.004
C01395=1185.942,-1.497,-44.582,-179.935,5.764,149.003
C01396=1185.936,-1.247,-44.596,-179.932,5.765,149.002
C01397=1185.931,-0.998,-44.610,-179.929,5.765,149.002
C01398=1185.926,-0.747,-44.623,-179.927,5.766,149.001
C01399=1185.921,-0.499,-44.637,-179.924,5.767,149.001
C01400=1185.916,-0.249,-44.651,-179.922,5.767,149.000
C01401=1185.911,0.001,-44.665,-179.920,5.768,149.000
C01402=1185.906,0.250,-44.678,-179.917,5.768,148.999
C01403=1185.901,0.500,-44.692,-179.914,5.769,148.998
C01404=1185.895,0.749,-44.705,-179.912,5.769,148.997
C01405=1185.890,0.999,-44.720,-179.909,5.770,148.997
C01406=1185.886,1.248,-44.733,-179.907,5.771,148.996
C01407=1185.880,1.498,-44.747,-179.904,5.771,148.996
C01408=1185.875,1.748,-44.761,-179.901,5.772,148.995
C01409=1185.870,1.998,-44.775,-179.899,5.773,148.994
C01410=1185.864,2.266,-44.790,-179.897,5.773,148.994
C01411=1185.859,2.536,-44.805,-179.894,5.774,148.993
C01412=1185.854,2.805,-44.819,-179.891,5.774,148.992
C01413=1185.849,3.074,-44.834,-179.889,5.774,148.992
C01414=1185.843,3.323,-44.848,-179.886,5.775,148.991
C01415=1185.838,3.573,-44.862,-179.883,5.775,148.990
C01416=1185.833,3.823,-44.876,-179.881,5.776,148.990
C01417=1185.827,4.072,-44.890,-179.879,5.777,148.989
C01418=1185.823,4.322,-44.903,-179.876,5.777,148.988
C01419=1185.818,4.571,-44.918,-179.874,5.778,148.988
C01420=1185.813,4.820,-44.932,-179.871,5.779,148.987
C01421=1185.807,5.071,-44.945,-179.868,5.779,148.987
C01422=1185.802,5.320,-44.959,-179.866,5.780,148.986
C01423=1185.798,5.570,-44.974,-179.864,5.780,148.986
C01424=1185.793,5.819,-44.987,-179.861,5.781,148.985
C01425=1185.788,6.068,-45.001,-179.858,5.781,148.984
C01426=1185.783,6.318,-45.016,-179.856,5.782,148.984
C01427=1185.777,6.568,-45.029,-179.853,5.783,148.983
C01428=1185.772,6.818,-45.043,-179.851,5.783,148.982
C01429=1185.767,7.067,-45.057,-179.848,5.784,148.982
C01430=1185.762,7.317,-45.072,-179.846,5.785,148.981
C01431=1185.756,7.566,-45.086,-179.843,5.785,148.980
C01432=1185.752,7.816,-45.100,-179.841,5.785,148.980
C01433=1185.747,8.065,-45.114,-179.838,5.786,148.979
C01434=1185.742,8.314,-45.127,-179.836,5.787,148.979
C01435=1185.737,8.564,-45.142,-179.833,5.787,148.978
C01436=1185.732,8.814,-45.156,-179.831,5.788,148.977
C01437=1185.727,9.063,-45.170,-179.828,5.789,148.977
C01438=1185.721,9.312,-45.184,-179.826,5.789,148.976
C01439=1185.716,9.563,-45.198,-179.823,5.790,148.975
C01440=1185.711,9.812,-45.212,-179.820,5.790,148.975
C01441=1185.706,10.062,-45.226,-179.818,5.791,148.974
C01442=1185.701,10.312,-45.241,-179.816,5.791,148.974
C01443=1185.696,10.561,-45.254,-179.813,5.792,148.973
C01444=1185.691,10.810,-45.269,-179.811,5.793,148.972
C01445=1185.686,11.060,-45.283,-179.808,5.793,148.972
C01446=1185.681,11.310,-45.297,-179.806,5.794,148.971
C01447=1185.675,11.559,-45.311,-179.803,5.794,148.970
C01448=1185.671,11.808,-45.326,-179.801,5.795,148.970
C01449=1185.666,12.058,-45.341,-179.798,5.796,148.969
C01450=1185.661,12.307,-45.355,-179.795,5.796,148.969
C01451=1185.656,12.557,-45.369,-179.793,5.797,148.968
C01452=1185.650,12.806,-45.383,-179.791,5.797,148.967
C01453=1185.645,13.056,-45.397,-179.788,5.798,148.967
C01454=1185.640,13.305,-45.412,-179.785,5.798,148.966
C01455=1185.635,13.555,-45.426,-179.783,5.799,148.966
C01456=1185.630,13.805,-45.440,-179.780,5.800,148.965
C01457=1185.625,14.055,-45.454,-179.778,5.800,148.964
C01458=1185.620,14.304,-45.468,-179.776,5.801,148.964
C01459=1185.615,14.553,-45.483,-179.773,5.802,148.963
C01460=1185.610,14.802,-45.498,-179.770,5.802,148.962
C01461=1185.605,15.052,-45.512,-179.768,5.803,148.962
C01462=1185.600,15.302,-45.526,-179.766,5.803,148.961
C01463=1185.595,15.552,-45.540,-179.763,5.804,148.961
C01464=1185.590,15.802,-45.555,-179.760,5.804,148.960
C01465=1185.584,16.051,-45.569,-179.758,5.805,148.959
C01466=1185.579,16.300,-45.584,-179.755,5.806,148.959
C01467=1185.575,16.549,-45.598,-179.753,5.806,148.958
C01468=1185.570,16.799,-45.613,-179.751,5.807,148.958
C01469=1185.565,17.049,-45.627,-179.747,5.808,148.957
C01470=1185.560,17.299,-45.641,-179.745,5.809,148.956
C01471=1185.555,17.548,-45.656,-179.742,5.809,148.956
C01472=1185.550,17.797,-45.671,-179.740,5.810,148.955
C01473=1185.544,18.047,-45.685,-179.737,5.811,148.954
C01474=1185.539,18.296,-45.699,-179.735,5.811,148.954
C01475=1185.534,18.545,-45.714,-179.732,5.812,148.953
C01476=1185.529,18.795,-45.729,-179.730,5.813,148.953
C01477=1185.524,19.045,-45.743,-179.727,5.813,148.952
C01478=1185.520,19.294,-45.758,-179.725,5.814,148.952
C01479=1185.514,19.544,-45.773,-179.722,5.814,148.951
C01480=1185.509,19.794,-45.787,-179.720,5.815,148.950
C01481=1185.504,20.043,-45.801,-179.717,5.815,148.949
C01482=1185.499,20.293,-45.816,-179.715,5.816,148.949
C01483=1185.494,20.542,-45.831,-179.712,5.817,148.948
C01484=1185.489,20.792,-45.845,-179.710,5.817,148.948
C01485=1185.483,21.041,-45.860,-179.707,5.818,148.947
C01486=1185.478,21.290,-45.874,-179.705,5.819,148.947
C01487=1185.474,21.539,-45.889,-179.702,5.819,148.946
C01488=1185.468,21.789,-45.904,-179.699,5.821,148.945
C01489=1185.463,22.039,-45.918,-179.697,5.821,148.945
C01490=1185.459,22.288,-45.933,-179.694,5.822,148.944
C01491=1185.454,22.538,-45.948,-179.691,5.822,148.943
C01492=1185.448,22.787,-45.963,-179.689,5.823,148.943
C01493=1185.443,23.037,-45.978,-179.687,5.824,148.942
C01494=1185.438,23.287,-45.992,-179.684,5.824,148.942
C01495=1185.434,23.536,-46.007,-179.682,5.825,148.941
C01496=1185.428,23.786,-46.022,-179.679,5.825,148.940
C01497=1185.423,24.035,-46.037,-179.677,5.826,148.940
C01498=1185.418,24.285,-46.051,-179.674,5.827,148.939
C01499=1185.414,24.534,-46.066,-179.672,5.827,148.939
C01500=1185.408,24.784,-46.081,-179.669,5.828,148.938
C01501=1185.403,25.033,-46.096,-179.666,5.829,148.937
C01502=1185.398,25.283,-46.110,-179.664,5.830,148.937
C01503=1185.393,25.532,-46.126,-179.661,5.830,148.936
C01504=1185.388,25.782,-46.140,-179.659,5.831,148.936
C01505=1185.383,26.031,-46.155,-179.656,5.832,148.935
C01506=1185.378,26.281,-46.170,-179.654,5.832,148.934
C01507=1185.373,26.530,-46.185,-179.651,5.833,148.934
C01508=1185.368,26.780,-46.199,-179.649,5.834,148.933
C01509=1185.363,27.029,-46.215,-179.646,5.834,148.932
C01510=1185.358,27.279,-46.229,-179.644,5.835,148.932
C01511=1185.352,27.528,-46.245,-179.641,5.836,148.931
C01512=1185.348,27.777,-46.260,-179.638,5.837,148.931
C01513=1185.343,28.027,-46.274,-179.635,5.837,148.930
C01514=1185.337,28.296,-46.290,-179.633,5.838,148.929
C01515=1185.332,28.564,-46.307,-179.631,5.839,148.929
C01516=1185.326,28.833,-46.323,-179.628,5.839,148.928
C01517=1185.321,29.102,-46.339,-179.625,5.841,148.928
C01518=1185.316,29.352,-46.354,-179.622,5.841,148.927
C01519=1185.311,29.602,-46.369,-179.620,5.841,148.926
C01520=1185.307,29.851,-46.384,-179.617,5.842,148.926
C01521=1185.301,30.100,-46.399,-179.615,5.843,148.925
C01522=1185.296,30.350,-46.414,-179.612,5.843,148.924
C01523=1185.291,30.600,-46.429,-179.610,5.844,148.924
C01524=1185.286,30.849,-46.444,-179.607,5.845,148.923
C01525=1185.281,31.099,-46.459,-179.604,5.846,148.923
C01526=1185.276,31.348,-46.474,-179.602,5.847,148.922
C01527=1185.271,31.597,-46.490,-179.599,5.847,148.921
C01528=1185.266,31.847,-46.504,-179.597,5.848,148.921
C01529=1185.261,32.097,-46.520,-179.594,5.849,148.920
C01530=1185.256,32.346,-46.535,-179.592,5.849,148.920
C01531=1185.251,32.595,-46.551,-179.589,5.850,148.919
C01532=1185.246,32.845,-46.565,-179.587,5.851,148.919
C01533=1185.241,33.095,-46.580,-179.584,5.852,148.918
C01534=1185.236,33.344,-46.595,-179.581,5.852,148.917
C01535=1185.230,33.593,-46.611,-179.579,5.853,148.917
C01536=1185.226,33.843,-46.626,-179.576,5.854,148.916
C01537=1185.221,34.093,-46.641,-179.574,5.854,148.915
C01538=1185.216,34.342,-46.656,-179.572,5.855,148.915
C01539=1185.211,34.591,-46.672,-179.569,5.856,148.914
C01540=1185.206,34.840,-46.687,-179.566,5.856,148.914
C01541=1185.201,35.090,-46.702,-179.563,5.858,148.913
C01542=1185.196,35.340,-46.717,-179.561,5.858,148.912
C01543=1185.191,35.590,-46.733,-179.558,5.859,148.912
C01544=1185.186,35.839,-46.748,-179.556,5.860,148.911
C01545=1185.181,36.088,-46.763,-179.553,5.860,148.911
C01546=1185.175,36.338,-46.779,-179.551,5.861,148.910
C01547=1185.171,36.587,-46.794,-179.549,5.862,148.910
C01548=1185.166,36.837,-46.810,-179.545,5.863,148.909
C01549=1185.161,37.086,-46.825,-179.543,5.864,148.908
C01550=1185.156,37.336,-46.840,-179.541,5.864,148.908
C01551=1185.150,37.585,-46.855,-179.538,5.865,148.907
C01552=1185.146,37.834,-46.870,-179.535,5.865,148.906
C01553=1185.141,38.084,-46.886,-179.533,5.866,148.906
C01554=1185.136,38.334,-46.902,-179.530,5.868,148.905
C01555=1185.131,38.583,-46.917,-179.527,5.868,148.905
C01556=1185.125,38.832,-46.932,-179.525,5.869,148.904
C01557=1185.120,39.082,-46.948,-179.522,5.869,148.903
C01558=1185.116,39.332,-46.963,-179.520,5.870,148.903
C01559=1185.111,39.581,-46.979,-179.518,5.871,148.902
C01560=1185.105,39.830,-46.994,-179.514,5.872,148.902
C01561=1185.101,40.079,-47.009,-179.512,5.873,148.901
C01562=1185.096,40.330,-47.025,-179.510,5.874,148.901
C01563=1185.090,40.579,-47.041,-179.507,5.874,148.900
C01564=1185.086,40.828,-47.056,-179.505,5.875,148.899
C01565=1185.080,41.077,-47.072,-179.502,5.875,148.899
C01566=1185.076,41.328,-47.087,-179.499,5.877,148.898
C01567=1185.070,41.577,-47.103,-179.497,5.878,148.898
C01568=1185.066,41.826,-47.118,-179.494,5.878,148.897
C01569=1185.060,42.075,-47.134,-179.492,5.879,148.896
C01570=1185.056,42.325,-47.150,-179.489,5.880,148.896
C01571=1185.050,42.574,-47.166,-179.487,5.880,148.895
C01572=1185.046,42.823,-47.181,-179.484,5.881,148.895
C01573=1185.041,43.074,-47.197,-179.481,5.882,148.894
C01574=1185.036,43.323,-47.212,-179.479,5.883,148.893
C01575=1185.030,43.572,-47.228,-179.477,5.884,148.893
C01576=1185.026,43.822,-47.243,-179.474,5.884,148.892
C01577=1185.021,44.072,-47.259,-179.471,5.885,148.892
C01578=1185.016,44.320,-47.275,-179.469,5.886,148.891
C01579=1185.010,44.570,-47.291,-179.466,5.887,148.891
C01580=1185.005,44.820,-47.307,-179.463,5.887,148.890
C01581=1185.001,45.069,-47.322,-179.461,5.888,148.889
C01582=1184.995,45.318,-47.337,-179.459,5.889,148.889
C01583=1184.991,45.568,-47.354,-179.455,5.890,148.888
C01584=1184.986,45.817,-47.370,-179.453,5.891,148.888
C01585=1184.980,46.067,-47.385,-179.450,5.891,148.887
C01586=1184.976,46.316,-47.401,-179.448,5.892,148.886
C01587=1184.971,46.566,-47.416,-179.446,5.893,148.886
C01588=1184.966,46.815,-47.433,-179.442,5.894,148.885
C01589=1184.961,47.065,-47.448,-179.440,5.895,148.885
C01590=1184.955,47.314,-47.464,-179.438,5.896,148.884
C01591=1184.951,47.564,-47.480,-179.435,5.896,148.883
C01592=1184.946,47.813,-47.496,-179.432,5.898,148.883
C01593=1184.941,48.062,-47.511,-179.430,5.898,148.882
C01594=1184.936,48.312,-47.527,-179.427,5.899,148.882
C01595=1184.931,48.561,-47.544,-179.425,5.900,148.881
C01596=1184.926,48.811,-47.559,-179.422,5.900,148.880
C01597=1184.921,49.060,-47.575,-179.420,5.902,148.880
C01598=1184.916,49.309,-47.591,-179.417,5.902,148.879
C01599=1184.911,49.559,-47.607,-179.414,5.903,148.879
C01600=1184.906,49.809,-47.623,-179.412,5.904,148.878
C01601=1184.901,50.058,-47.640,-179.409,5.904,148.878
C01602=1184.896,50.308,-47.655,-179.406,5.906,148.877
C01603=1184.891,50.556,-47.671,-179.404,5.907,148.876
C01604=1184.887,50.806,-47.687,-179.401,5.907,148.876
C01605=1184.881,51.056,-47.702,-179.399,5.908,148.875
C01606=1184.877,51.305,-47.719,-179.396,5.909,148.875
C01607=1184.871,51.555,-47.735,-179.393,5.910,148.874
C01608=1184.867,51.804,-47.751,-179.391,5.911,148.874
C01609=1184.862,52.053,-47.767,-179.389,5.911,148.873
C01610=1184.857,52.304,-47.783,-179.386,5.913,148.872
C01611=1184.852,52.552,-47.799,-179.383,5.913,148.872
C01612=1184.846,52.802,-47.815,-179.381,5.914,148.871
C01613=1184.842,53.051,-47.831,-179.378,5.915,148.871
C01614=1184.836,53.301,-47.847,-179.375,5.916,148.870
C01615=1184.832,53.550,-47.864,-179.373,5.917,148.869
C01616=1184.827,53.799,-47.879,-179.370,5.918,148.869
C01617=1184.822,54.049,-47.896,-179.368,5.918,148.868
C01618=1184.817,54.317,-47.913,-179.365,5.919,148.868
C01619=1184.811,54.586,-47.930,-179.362,5.920,148.867
C01620=1184.806,54.855,-47.949,-179.359,5.922,148.867
C01621=1184.800,55.123,-47.966,-179.357,5.922,148.866
C01622=1184.795,55.372,-47.982,-179.354,5.923,148.865
C01623=1184.790,55.622,-47.998,-179.352,5.924,148.865
C01624=1184.785,55.871,-48.014,-179.349,5.925,148.864
C01625=1184.780,56.121,-48.030,-179.346,5.926,148.864
C01626=1184.775,56.370,-48.047,-179.344,5.926,148.863
C01627=1184.771,56.619,-48.063,-179.341,5.927,148.862
C01628=1184.765,56.869,-48.079,-179.338,5.929,148.862
C01629=1184.761,57.118,-48.095,-179.336,5.929,148.861
C01630=1184.755,57.369,-48.112,-179.334,5.930,148.861
C01631=1184.750,57.617,-48.128,-179.330,5.931,148.860
C01632=1184.746,57.867,-48.145,-179.328,5.932,148.859
C01633=1184.740,58.116,-48.161,-179.326,5.933,148.859
C01634=1184.736,58.366,-48.177,-179.323,5.933,148.858
C01635=1184.731,58.615,-48.194,-179.320,5.935,148.858
C01636=1184.726,58.865,-48.210,-179.318,5.935,148.857
C01637=1184.721,59.113,-48.226,-179.315,5.936,148.857
C01638=1184.716,59.363,-48.243,-179.313,5.937,148.856
C01639=1184.710,59.613,-48.259,-179.310,5.938,148.855
C01640=1184.706,59.862,-48.275,-179.308,5.939,148.855
C01641=1184.701,60.112,-48.292,-179.305,5.940,148.854
C01642=1184.696,60.360,-48.308,-179.302,5.941,148.854
C01643=1184.691,60.611,-48.325,-179.300,5.942,148.853
C01644=1184.686,60.860,-48.341,-179.297,5.942,148.853
C01645=1184.681,61.109,-48.358,-179.295,5.943,148.852
C01646=1184.677,61.359,-48.374,-179.292,5.945,148.852
C01647=1184.672,61.607,-48.391,-179.289,5.945,148.851
C01648=1184.666,61.858,-48.407,-179.287,5.946,148.850
C01649=1184.661,62.107,-48.424,-179.284,5.947,148.850
C01650=1184.657,62.356,-48.440,-179.281,5.948,148.849
C01651=1184.652,62.605,-48.457,-179.279,5.949,148.849
C01652=1184.646,62.855,-48.474,-179.276,5.950,148.848
C01653=1184.641,63.105,-48.490,-179.273,5.951,148.848
C01654=1184.637,63.354,-48.507,-179.271,5.952,148.847
C01655=1184.632,63.603,-48.523,-179.269,5.952,148.846
C01656=1184.627,63.853,-48.540,-179.265,5.954,148.846
C01657=1184.622,64.102,-48.556,-179.263,5.955,148.845
C01658=1184.617,64.351,-48.573,-179.261,5.955,148.845
C01659=1184.612,64.601,-48.590,-179.258,5.957,148.844
C01660=1184.607,64.850,-48.607,-179.255,5.957,148.844
C01661=1184.602,65.100,-48.623,-179.253,5.958,148.843
C01662=1184.598,65.349,-48.639,-179.250,5.960,148.843
C01663=1184.592,65.598,-48.656,-179.247,5.960,148.842
C01664=1184.587,65.848,-48.673,-179.245,5.961,148.841
C01665=1184.583,66.097,-48.689,-179.242,5.962,148.841
C01666=1184.577,66.346,-48.706,-179.240,5.963,148.840
C01667=1184.572,66.596,-48.723,-179.237,5.964,148.840
C01668=1184.568,66.845,-48.740,-179.234,5.965,148.839
C01669=1184.562,67.094,-48.757,-179.232,5.966,148.839
C01670=1184.558,67.344,-48.773,-179.230,5.967,148.838
C01671=1184.552,67.594,-48.791,-179.227,5.967,148.837
C01672=1184.548,67.843,-48.807,-179.224,5.969,148.837
C01673=1184.543,68.092,-48.824,-179.222,5.970,148.836
C01674=1184.538,68.342,-48.841,-179.219,5.970,148.836
C01675=1184.533,68.591,-48.857,-179.216,5.972,148.835
C01676=1184.528,68.840,-48.874,-179.214,5.972,148.835
C01677=1184.523,69.090,-48.891,-179.211,5.973,148.834
C01678=1184.518,69.339,-48.908,-179.208,5.975,148.834
C01679=1184.514,69.588,-48.926,-179.206,5.976,148.833
C01680=1184.508,69.837,-48.942,-179.204,5.976,148.832
C01681=1184.503,70.087,-48.959,-179.200,5.977,148.832
C01682=1184.499,70.337,-48.976,-179.198,5.978,148.831
C01683=1184.494,70.586,-48.993,-179.195,5.980,148.831
C01684=1184.488,70.835,-49.009,-179.193,5.981,148.830
C01685=1184.484,71.085,-49.026,-179.190,5.981,148.830
C01686=1184.479,71.334,-49.043,-179.187,5.983,148.829
C01687=1184.475,71.583,-49.061,-179.185,5.983,148.829
C01688=1184.469,71.832,-49.078,-179.183,5.984,148.828
C01689=1184.464,72.082,-49.094,-179.179,5.986,148.827
C01690=1184.459,72.332,-49.112,-179.177,5.987,148.827
C01691=1184.455,72.581,-49.128,-179.175,5.987,148.826
C01692=1184.449,72.831,-49.146,-179.171,5.988,148.826
C01693=1184.445,73.079,-49.163,-179.169,5.989,148.825
C01694=1184.439,73.329,-49.180,-179.167,5.990,148.825
C01695=1184.435,73.578,-49.197,-179.164,5.992,148.824
C01696=1184.430,73.828,-49.214,-179.161,5.992,148.824
C01697=1184.426,74.077,-49.231,-179.159,5.994,148.823
C01698=1184.420,74.326,-49.248,-179.156,5.994,148.822
C01699=1184.414,74.576,-49.265,-179.154,5.995,148.822
C01700=1184.410,74.825,-49.282,-179.151,5.997,148.821
C01701=1184.405,75.075,-49.300,-179.148,5.997,148.821
C01702=1184.401,75.324,-49.317,-179.146,5.998,148.820
C01703=1184.395,75.574,-49.334,-179.143,6.000,148.820
C01704=1184.391,75.822,-49.351,-179.141,6.000,148.819
C01705=1184.385,76.072,-49.368,-179.138,6.002,148.819
C01706=1184.380,76.322,-49.385,-179.135,6.003,148.818
C01707=1184.376,76.570,-49.403,-179.133,6.003,148.818
C01708=1184.371,76.820,-49.420,-179.130,6.005,148.817
C01709=1184.366,77.070,-49.437,-179.127,6.005,148.816
C01710=1184.361,77.319,-49.455,-179.125,6.006,148.816
C01711=1184.356,77.568,-49.472,-179.122,6.008,148.815
C01712=1184.351,77.817,-49.488,-179.120,6.008,148.815
C01713=1184.346,78.067,-49.506,-179.116,6.010,148.814
C01714=1184.341,78.316,-49.524,-179.114,6.011,148.814
C01715=1184.337,78.565,-49.541,-179.112,6.011,148.813
C01716=1184.332,78.815,-49.558,-179.109,6.013,148.813
C01717=1184.327,79.064,-49.576,-179.106,6.014,148.812
C01718=1184.322,79.314,-49.593,-179.104,6.015,148.812
C01719=1184.317,79.564,-49.610,-179.101,6.016,148.811
C01720=1184.311,79.812,-49.628,-179.099,6.017,148.811
C01721=1184.307,80.062,-49.644,-179.096,6.018,148.810
C01722=1184.302,80.330,-49.664,-179.094,6.019,148.809
C01723=1184.297,80.599,-49.683,-179.090,6.020,148.809
C01724=1184.291,80.867,-49.702,-179.087,6.022,148.808
C01725=1184.285,81.135,-49.720,-179.085,6.023,148.808
C01726=1184.281,81.385,-49.737,-179.082,6.024,148.807
C01727=1184.276,81.634,-49.755,-179.080,6.025,148.807
C01728=1184.271,81.883,-49.773,-179.077,6.025,148.806
C01729=1184.266,82.133,-49.790,-179.074,6.027,148.806
C01730=1184.262,82.382,-49.808,-179.072,6.028,148.805
C01731=1184.257,82.631,-49.825,-179.069,6.029,148.805
C01732=1184.252,82.881,-49.843,-179.066,6.030,148.804
C01733=1184.246,83.130,-49.860,-179.064,6.031,148.803
C01734=1184.241,83.380,-49.878,-179.061,6.032,148.803
C01735=1184.237,83.628,-49.895,-179.059,6.033,148.802
C01736=1184.232,83.878,-49.913,-179.056,6.034,148.802
C01737=1184.227,84.127,-49.931,-179.053,6.035,148.801
C01738=1184.222,84.377,-49.948,-179.050,6.037,148.801
C01739=1184.217,84.626,-49.966,-179.048,6.038,148.800
C01740=1184.213,84.875,-49.983,-179.046,6.038,148.800
C01741=1184.208,85.125,-50.001,-179.043,6.040,148.799
C01742=1184.203,85.374,-50.019,-179.040,6.040,148.798
C01743=1184.198,85.623,-50.036,-179.037,6.042,148.798
C01744=1184.193,85.872,-50.054,-179.035,6.043,148.797
C01745=1184.188,86.122,-50.072,-179.032,6.044,148.797
C01746=1184.184,86.371,-50.089,-179.029,6.045,148.796
C01747=1184.179,86.620,-50.107,-179.027,6.047,148.796
C01748=1184.173,86.870,-50.124,-179.024,6.047,148.795
C01749=1184.168,87.119,-50.142,-179.022,6.048,148.795
C01750=1184.164,87.368,-50.160,-179.019,6.049,148.794
C01751=1184.159,87.618,-50.178,-179.017,6.050,148.794
C01752=1184.153,87.867,-50.196,-179.013,6.052,148.793
C01753=1184.149,88.117,-50.214,-179.011,6.053,148.793
C01754=1184.144,88.366,-50.232,-179.008,6.054,148.792
C01755=1184.139,88.615,-50.250,-179.006,6.055,148.792
C01756=1184.135,88.864,-50.267,-179.003,6.057,148.791
C01757=1184.129,89.114,-50.284,-179.001,6.057,148.791
C01758=1184.124,89.363,-50.302,-178.998,6.059,148.790
C01759=1184.120,89.613,-50.320,-178.995,6.059,148.790
C01760=1184.115,89.862,-50.338,-178.993,6.060,148.789
C01761=1184.110,90.111,-50.356,-178.990,6.062,148.788
C01762=1184.105,90.360,-50.374,-178.988,6.063,148.788
C01763=1184.100,90.609,-50.392,-178.985,6.064,148.787
C01764=1184.096,90.859,-50.410,-178.982,6.065,148.787
C01765=1184.090,91.108,-50.428,-178.979,6.066,148.786
C01766=1184.085,91.358,-50.446,-178.977,6.067,148.786
C01767=1184.080,91.607,-50.464,-178.974,6.068,148.785
C01768=1184.076,91.856,-50.482,-178.972,6.069,148.785
C01769=1184.071,92.106,-50.500,-178.969,6.071,148.784
C01770=1184.066,92.355,-50.518,-178.966,6.072,148.784
C01771=1184.061,92.604,-50.536,-178.964,6.073,148.783
C01772=1184.057,92.853,-50.554,-178.961,6.074,148.783
C01773=1184.052,93.102,-50.572,-178.958,6.076,148.782
C01774=1184.047,93.352,-50.590,-178.956,6.076,148.782
C01775=1184.042,93.601,-50.608,-178.953,6.078,148.781
C01776=1184.037,93.851,-50.627,-178.950,6.078,148.781
C01777=1184.032,94.100,-50.645,-178.948,6.080,148.780
C01778=1184.027,94.349,-50.663,-178.946,6.081,148.780
C01779=1184.022,94.599,-50.681,-178.942,6.082,148.779
C01780=1184.017,94.848,-50.699,-178.940,6.083,148.779
C01781=1184.012,95.097,-50.717,-178.937,6.085,148.778
C01782=1184.008,95.347,-50.735,-178.935,6.086,148.778
C01783=1184.003,95.596,-50.753,-178.932,6.087,148.777
C01784=1183.998,95.845,-50.771,-178.930,6.088,148.777
C01785=1183.993,96.094,-50.789,-178.926,6.089,148.776
C01786=1183.988,96.343,-50.808,-178.924,6.090,148.775
C01787=1183.983,96.592,-50.826,-178.922,6.092,148.775
C01788=1183.979,96.842,-50.845,-178.919,6.093,148.774
C01789=1183.974,97.091,-50.863,-178.916,6.094,148.774
C01790=1183.969,97.341,-50.881,-178.914,6.095,148.773
C01791=1183.964,97.590,-50.898,-178.911,6.097,148.773
C01792=1183.959,97.840,-50.917,-178.908,6.097,148.772
C01793=1183.954,98.088,-50.936,-178.906,6.099,148.772
C01794=1183.949,98.338,-50.954,-178.903,6.100,148.771
C01795=1183.944,98.587,-50.972,-178.900,6.101,148.771
C01796=1183.939,98.836,-50.990,-178.898,6.102,148.770
C01797=1183.935,99.086,-51.008,-178.895,6.103,148.770
C01798=1183.930,99.335,-51.028,-178.893,6.104,148.769
C01799=1183.925,99.584,-51.046,-178.890,6.106,148.769
C01800=1183.920,99.833,-51.064,-178.887,6.107,148.768
C01801=1183.916,100.083,-51.082,-178.885,6.108,148.768
C01802=1183.910,100.332,-51.101,-178.882,6.109,148.767
C01803=1183.905,100.581,-51.119,-178.879,6.111,148.767
C01804=1183.901,100.831,-51.138,-178.877,6.112,148.766
C01805=1183.896,101.080,-51.156,-178.874,6.113,148.766
C01806=1183.891,101.329,-51.175,-178.871,6.115,148.765
C01807=1183.886,101.578,-51.193,-178.869,6.115,148.765
C01808=1183.882,101.828,-51.211,-178.866,6.117,148.764
C01809=1183.877,102.077,-51.230,-178.863,6.117,148.764
C01810=1183.871,102.326,-51.248,-178.861,6.119,148.763
C01811=1183.867,102.576,-51.267,-178.859,6.120,148.763
C01812=1183.862,102.824,-51.286,-178.855,6.121,148.762
C01813=1183.857,103.074,-51.304,-178.853,6.122,148.762
C01814=1183.852,103.323,-51.322,-178.850,6.124,148.761
C01815=1183.848,103.572,-51.341,-178.847,6.126,148.761
C01816=1183.842,103.822,-51.360,-178.845,6.126,148.760
C01817=1183.838,104.070,-51.378,-178.842,6.128,148.760
C01818=1183.833,104.320,-51.397,-178.840,6.129,148.759
C01819=1183.828,104.570,-51.415,-178.837,6.130,148.759
C01820=1183.823,104.818,-51.434,-178.835,6.131,148.758
C01821=1183.819,105.068,-51.452,-178.832,6.133,148.758
C01822=1183.813,105.317,-51.472,-178.829,6.133,148.757
C01823=1183.809,105.567,-51.490,-178.827,6.135,148.757
C01824=1183.804,105.816,-51.509,-178.824,6.137,148.756
C01825=1183.799,106.065,-51.527,-178.821,6.137,148.756
C01826=1183.794,106.334,-51.548,-178.818,6.139,148.755
C01827=1183.789,106.602,-51.568,-178.815,6.140,148.755
C01828=1183.783,106.870,-51.588,-178.813,6.141,148.754
C01829=1183.779,107.139,-51.608,-178.810,6.143,148.754
C01830=1183.773,107.388,-51.627,-178.807,6.144,148.753
C01831=1183.769,107.637,-51.646,-178.805,6.145,148.753
C01832=1183.764,107.886,-51.665,-178.802,6.147,148.752
C01833=1183.759,108.136,-51.683,-178.799,6.148,148.752
C01834=1183.754,108.384,-51.702,-178.797,6.149,148.751
C01835=1183.749,108.634,-51.721,-178.794,6.151,148.751
C01836=1183.744,108.883,-51.740,-178.791,6.151,148.750
C01837=1183.740,109.133,-51.758,-178.789,6.153,148.750
C01838=1183.734,109.382,-51.778,-178.786,6.154,148.749
C01839=1183.730,109.631,-51.797,-178.783,6.155,148.749
